C01785=1032.766,450.226,-154.652,176.488,48.489,160.264
C01786=1032.794,450.472,-154.693,176.509,48.493,160.268
C01787=1032.823,450.716,-154.734,176.528,48.497,160.272
C01788=1032.851,450.962,-154.775,176.549,48.502,160.277
C01789=1032.882,451.208,-154.815,176.569,48.506,160.281
C01790=1032.912,451.453,-154.855,176.590,48.510,160.285
C01791=1032.942,451.698,-154.894,176.611,48.514,160.290
C01792=1032.973,451.944,-154.933,176.632,48.519,160.294
C01793=1033.006,452.191,-154.972,176.652,48.523,160.299
C01794=1033.037,452.435,-155.009,176.673,48.527,160.303
C01795=1033.070,452.681,-155.047,176.695,48.530,160.307
C01796=1033.104,452.933,-155.086,176.716,48.534,160.312
C01797=1033.139,453.185,-155.123,176.737,48.538,160.316
C01798=1032.855,453.248,-155.453,176.741,48.604,160.337
C01799=1032.824,453.021,-155.419,176.721,48.600,160.333
C01800=1032.792,452.792,-155.385,176.702,48.597,160.329
C01801=1032.760,452.547,-155.347,176.680,48.593,160.325
C01802=1032.728,452.301,-155.309,176.659,48.589,160.320
C01803=1032.695,452.056,-155.271,176.639,48.585,160.316
C01804=1032.664,451.810,-155.232,176.617,48.582,160.312
C01805=1032.633,451.564,-155.193,176.596,48.578,160.307
C01806=1032.603,451.319,-155.154,176.577,48.573,160.303
C01807=1032.573,451.074,-155.114,176.556,48.569,160.299
C01808=1032.543,450.827,-155.074,176.535,48.566,160.294
C01809=1032.514,450.583,-155.033,176.515,48.561,160.290
C01810=1032.486,450.338,-154.992,176.494,48.557,160.286
C01811=1032.458,450.092,-154.950,176.474,48.552,160.281
C01812=1032.431,449.847,-154.908,176.454,48.548,160.277
C01813=1032.404,449.602,-154.865,176.434,48.543,160.273
C01814=1032.377,449.357,-154.823,176.414,48.539,160.268
C01815=1032.351,449.112,-154.779,176.394,48.534,160.264
C01816=1032.326,448.866,-154.736,176.374,48.530,160.259
C01817=1032.301,448.622,-154.691,176.355,48.524,160.255
C01818=1032.276,448.377,-154.647,176.334,48.519,160.250
C01819=1032.252,448.131,-154.602,176.316,48.515,160.246
C01820=1032.229,447.887,-154.556,176.296,48.510,160.242
C01821=1032.206,447.643,-154.511,176.276,48.504,160.237
C01822=1032.183,447.398,-154.465,176.258,48.499,160.233
C01823=1032.162,447.153,-154.418,176.238,48.494,160.228
C01824=1032.140,446.909,-154.371,176.219,48.489,160.224
C01825=1032.119,446.665,-154.324,176.200,48.483,160.220
C01826=1032.099,446.420,-154.276,176.181,48.478,160.215
C01827=1032.079,446.176,-154.227,176.162,48.472,160.211
C01828=1032.060,445.932,-154.179,176.143,48.467,160.206
C01829=1032.041,445.688,-154.130,176.124,48.461,160.201
C01830=1032.022,445.444,-154.080,176.106,48.455,160.197
C01831=1032.004,445.200,-154.030,176.088,48.449,160.193
C01832=1031.987,444.957,-153.980,176.069,48.443,160.188
C01833=1031.969,444.713,-153.928,176.050,48.437,160.183
C01834=1031.953,444.468,-153.878,176.033,48.431,160.179
C01835=1031.938,444.225,-153.826,176.014,48.425,160.174
C01836=1031.921,443.982,-153.774,175.996,48.419,160.170
C01837=1031.908,443.739,-153.721,175.977,48.412,160.165
C01838=1031.892,443.495,-153.668,175.960,48.406,160.161
C01839=1031.879,443.253,-153.615,175.942,48.399,160.156
C01840=1031.864,443.010,-153.562,175.924,48.393,160.152
C01841=1031.851,442.766,-153.509,175.906,48.386,160.147
C01842=1031.838,442.521,-153.455,175.889,48.379,160.142
C01843=1031.824,442.278,-153.402,175.870,48.374,160.138
C01844=1031.810,442.034,-153.348,175.853,48.367,160.133
C01845=1031.796,441.790,-153.296,175.836,48.361,160.129
C01846=1031.783,441.546,-153.242,175.818,48.354,160.125
C01847=1031.769,441.302,-153.190,175.801,48.347,160.120
C01848=1031.755,441.058,-153.136,175.784,48.341,160.116
C01849=1031.742,440.814,-153.084,175.766,48.335,160.111
C01850=1031.728,440.570,-153.030,175.749,48.329,160.107
C01851=1031.715,440.326,-152.977,175.732,48.322,160.103
C01852=1031.702,440.082,-152.925,175.715,48.316,160.098
C01853=1031.688,439.838,-152.871,175.698,48.310,160.094
C01854=1031.675,439.594,-152.820,175.681,48.304,160.090
C01855=1031.662,439.350,-152.766,175.664,48.297,160.085
C01856=1031.648,439.106,-152.714,175.646,48.291,160.081
C01857=1031.634,438.844,-152.657,175.629,48.284,160.076
C01858=1031.620,438.582,-152.601,175.611,48.278,160.072
C01859=1031.606,438.319,-152.544,175.593,48.271,160.067
C01860=1031.591,438.057,-152.489,175.575,48.265,160.063
C01861=1031.578,437.813,-152.436,175.559,48.258,160.059
C01862=1031.565,437.569,-152.385,175.542,48.253,160.054
C01863=1031.552,437.324,-152.332,175.526,48.246,160.050
C01864=1031.539,437.080,-152.280,175.509,48.241,160.046
C01865=1031.526,436.836,-152.228,175.494,48.234,160.042
C01866=1031.513,436.592,-152.176,175.477,48.229,160.038
C01867=1031.500,436.347,-152.124,175.461,48.222,160.034
C01868=1031.487,436.103,-152.072,175.444,48.217,160.030
C01869=1031.474,435.859,-152.021,175.429,48.211,160.026
C01870=1031.462,435.615,-151.969,175.413,48.205,160.022
C01871=1031.448,435.370,-151.917,175.396,48.199,160.018
C01872=1031.436,435.126,-151.866,175.381,48.193,160.014
C01873=1031.423,434.882,-151.814,175.365,48.187,160.010
C01874=1031.410,434.637,-151.763,175.350,48.182,160.006
C01875=1031.398,434.392,-151.711,175.334,48.176,160.002
C01876=1031.385,434.149,-151.660,175.317,48.170,159.998
C01877=1031.366,433.797,-151.586,175.296,48.162,159.992
C01878=1031.348,433.447,-151.513,175.273,48.154,159.987
C01879=1031.330,433.095,-151.440,175.251,48.145,159.981
C01880=1031.312,432.744,-151.366,175.229,48.137,159.976
C01881=1031.299,432.500,-151.315,175.214,48.132,159.972
C01882=1031.287,432.256,-151.265,175.198,48.126,159.968
C01883=1031.274,432.011,-151.214,175.183,48.121,159.965
C01884=1031.262,431.766,-151.163,175.168,48.115,159.961
C01885=1031.249,431.521,-151.112,175.153,48.110,159.957
C01886=1031.237,431.277,-151.062,175.137,48.104,159.953
C01887=1031.224,431.032,-151.011,175.123,48.098,159.950
C01888=1031.212,430.788,-150.961,175.108,48.093,159.946
C01889=1031.199,430.543,-150.910,175.093,48.087,159.942
C01890=1031.187,430.299,-150.860,175.078,48.082,159.938
C01891=1031.175,430.054,-150.809,175.064,48.077,159.935
C01892=1031.163,429.809,-150.758,175.049,48.071,159.931
C01893=1031.151,429.565,-150.709,175.033,48.066,159.928
C01894=1031.139,429.320,-150.659,175.019,48.061,159.924
C01895=1031.126,429.076,-150.608,175.004,48.055,159.920
C01896=1031.114,428.831,-150.558,174.990,48.050,159.917
C01897=1031.102,428.586,-150.507,174.976,48.045,159.913
C01898=1031.091,428.342,-150.457,174.961,48.039,159.910
C01899=1031.078,428.097,-150.407,174.946,48.034,159.906
C01900=1031.066,427.852,-150.357,174.933,48.029,159.903
C01901=1031.055,427.608,-150.308,174.919,48.023,159.899
C01902=1031.042,427.363,-150.258,174.904,48.019,159.896
C01903=1031.030,427.118,-150.208,174.890,48.013,159.892
C01904=1031.019,426.874,-150.158,174.876,48.008,159.889
C01905=1031.007,426.628,-150.108,174.861,48.003,159.885
C01906=1030.995,426.383,-150.058,174.847,47.998,159.882
C01907=1030.983,426.139,-150.009,174.834,47.993,159.878
C01908=1030.971,425.893,-149.960,174.819,47.988,159.875
C01909=1030.959,425.649,-149.911,174.805,47.983,159.872
C01910=1030.947,425.404,-149.861,174.791,47.978,159.868
C01911=1030.935,425.159,-149.812,174.778,47.972,159.865
C01912=1030.923,424.914,-149.762,174.764,47.967,159.861
C01913=1030.913,424.705,-149.720,174.752,47.963,159.859
C01914=1030.903,424.497,-149.678,174.740,47.959,159.856
C01915=1030.893,424.288,-149.636,174.729,47.955,159.853
C01916=1030.883,424.079,-149.594,174.717,47.950,159.850
C01917=1030.874,423.871,-149.553,174.706,47.947,159.847
C01918=1030.864,423.662,-149.511,174.693,47.942,159.845
C01919=1030.854,423.453,-149.469,174.682,47.938,159.842
C01920=1030.844,423.244,-149.428,174.671,47.934,159.839
C01921=1030.833,422.999,-149.379,174.657,47.929,159.836
C01922=1030.821,422.753,-149.330,174.644,47.924,159.833
C01923=1030.809,422.509,-149.280,174.630,47.920,159.829
C01924=1030.797,422.264,-149.233,174.617,47.914,159.826
C01925=1030.786,422.019,-149.184,174.604,47.910,159.823
C01926=1030.775,421.773,-149.135,174.591,47.905,159.820
C01927=1030.763,421.529,-149.087,174.578,47.900,159.817
C01928=1030.751,421.283,-149.038,174.564,47.896,159.813
C01929=1030.740,421.038,-148.989,174.551,47.891,159.810
C01930=1030.729,420.793,-148.941,174.539,47.886,159.807
C01931=1030.717,420.548,-148.893,174.525,47.882,159.804
C01932=1030.705,420.303,-148.844,174.512,47.877,159.801
C01933=1030.695,420.058,-148.796,174.499,47.872,159.798
C01934=1030.683,419.813,-148.749,174.486,47.867,159.795
C01935=1030.672,419.568,-148.700,174.473,47.863,159.792
C01936=1030.661,419.323,-148.652,174.461,47.858,159.789
C01937=1030.649,419.078,-148.604,174.447,47.854,159.786
C01938=1030.638,418.832,-148.556,174.434,47.850,159.783
C01939=1030.627,418.587,-148.508,174.422,47.845,159.779
C01940=1030.616,418.342,-148.461,174.409,47.841,159.777
C01941=1030.604,418.097,-148.412,174.397,47.836,159.773
C01942=1030.593,417.852,-148.364,174.384,47.831,159.771
C01943=1030.582,417.607,-148.317,174.372,47.827,159.768
C01944=1030.571,417.361,-148.269,174.359,47.822,159.765
C01945=1030.560,417.116,-148.221,174.346,47.818,159.762
C01946=1030.549,416.872,-148.173,174.334,47.814,159.759
C01947=1030.538,416.626,-148.126,174.322,47.809,159.756
C01948=1030.527,416.380,-148.077,174.310,47.805,159.753
C01949=1030.516,416.135,-148.031,174.298,47.801,159.750
C01950=1030.505,415.890,-147.983,174.285,47.796,159.747
C01951=1030.494,415.645,-147.936,174.273,47.792,159.744
C01952=1030.483,415.399,-147.889,174.261,47.788,159.741
C01953=1030.472,415.154,-147.842,174.248,47.783,159.739
C01954=1030.461,414.909,-147.794,174.236,47.780,159.736
C01955=1030.450,414.664,-147.747,174.224,47.775,159.733
C01956=1030.439,414.418,-147.700,174.212,47.771,159.730
C01957=1030.428,414.173,-147.653,174.199,47.767,159.727
C01958=1030.418,413.928,-147.606,174.187,47.763,159.725
C01959=1030.406,413.682,-147.559,174.175,47.758,159.722
C01960=1030.396,413.437,-147.512,174.164,47.754,159.719
C01961=1030.385,413.192,-147.465,174.152,47.750,159.716
C01962=1030.374,412.947,-147.419,174.140,47.746,159.713
C01963=1030.363,412.701,-147.371,174.128,47.742,159.711
C01964=1030.352,412.456,-147.324,174.116,47.737,159.708
C01965=1030.343,412.210,-147.278,174.105,47.733,159.705
C01966=1030.332,411.965,-147.231,174.093,47.730,159.703
C01967=1030.321,411.720,-147.185,174.082,47.726,159.700
C01968=1030.310,411.473,-147.138,174.070,47.722,159.697
C01969=1030.299,411.229,-147.091,174.058,47.717,159.694
C01970=1030.289,410.983,-147.044,174.046,47.713,159.692
C01971=1030.278,410.738,-146.998,174.035,47.709,159.689
C01972=1030.268,410.492,-146.951,174.023,47.705,159.686
C01973=1030.258,410.247,-146.905,174.012,47.702,159.684
C01974=1030.247,410.001,-146.859,174.000,47.698,159.681
C01975=1030.236,409.756,-146.813,173.989,47.694,159.679
C01976=1030.226,409.510,-146.767,173.977,47.690,159.676
C01977=1030.215,409.241,-146.716,173.965,47.686,159.673
C01978=1030.203,408.972,-146.666,173.952,47.682,159.670
C01979=1030.191,408.703,-146.615,173.940,47.677,159.668
C01980=1030.180,408.433,-146.565,173.928,47.674,159.665
C01981=1030.169,408.188,-146.519,173.916,47.670,159.662
C01982=1030.158,407.942,-146.473,173.906,47.666,159.660
C01983=1030.148,407.696,-146.428,173.894,47.662,159.657
C01984=1030.137,407.451,-146.382,173.883,47.659,159.655
C01985=1030.127,407.205,-146.336,173.871,47.655,159.652
C01986=1030.117,406.960,-146.290,173.861,47.651,159.650
C01987=1030.106,406.715,-146.244,173.850,47.648,159.647
C01988=1030.096,406.468,-146.198,173.838,47.644,159.645
C01989=1030.086,406.223,-146.153,173.828,47.640,159.642
C01990=1030.076,405.978,-146.107,173.817,47.637,159.640
C01991=1030.065,405.732,-146.062,173.806,47.633,159.637
C01992=1030.055,405.487,-146.016,173.795,47.629,159.635
C01993=1030.045,405.240,-145.971,173.784,47.626,159.633
C01994=1030.035,404.996,-145.926,173.773,47.622,159.630
C01995=1030.025,404.749,-145.880,173.762,47.619,159.628
C01996=1030.015,404.504,-145.835,173.752,47.615,159.625
C01997=1030.004,404.258,-145.790,173.741,47.612,159.623
C01998=1029.994,404.013,-145.744,173.730,47.608,159.620
C01999=1029.984,403.767,-145.699,173.719,47.605,159.618
C02000=1029.974,403.522,-145.654,173.709,47.601,159.616
C02001=1029.964,403.276,-145.608,173.699,47.598,159.613
C02002=1029.954,403.031,-145.563,173.688,47.594,159.611
C02003=1029.944,402.785,-145.519,173.677,47.590,159.609
C02004=1029.934,402.539,-145.473,173.666,47.588,159.606
C02005=1029.924,402.293,-145.429,173.656,47.584,159.604
C02006=1029.915,402.048,-145.384,173.646,47.581,159.602
C02007=1029.904,401.802,-145.339,173.635,47.577,159.599
C02008=1029.894,401.556,-145.294,173.625,47.574,159.597
C02009=1029.885,401.311,-145.249,173.615,47.570,159.595
C02010=1029.874,401.064,-145.204,173.604,47.567,159.593
C02011=1029.865,400.819,-145.159,173.594,47.564,159.590
C02012=1029.855,400.573,-145.114,173.583,47.560,159.588
C02013=1029.846,400.327,-145.070,173.573,47.557,159.586
C02014=1029.835,400.082,-145.026,173.563,47.554,159.584
C02015=1029.825,399.836,-144.981,173.552,47.550,159.581
C02016=1029.815,399.590,-144.936,173.542,47.547,159.579
C02017=1029.806,399.344,-144.892,173.531,47.544,159.577
C02018=1029.795,399.099,-144.847,173.521,47.541,159.575
C02019=1029.786,398.853,-144.803,173.512,47.538,159.572
C02020=1029.776,398.607,-144.758,173.502,47.535,159.570
C02021=1029.767,398.361,-144.714,173.492,47.532,159.568
C02022=1029.757,398.115,-144.671,173.482,47.528,159.566
C02023=1029.747,397.870,-144.626,173.471,47.525,159.564
C02024=1029.737,397.624,-144.582,173.461,47.523,159.562
C02025=1029.727,397.378,-144.538,173.451,47.520,159.560
C02026=1029.718,397.132,-144.494,173.441,47.516,159.557
C02027=1029.707,396.886,-144.450,173.431,47.513,159.555
C02028=1029.698,396.640,-144.406,173.422,47.510,159.553
C02029=1029.689,396.394,-144.362,173.412,47.507,159.551
C02030=1029.678,396.148,-144.318,173.402,47.504,159.549
C02031=1029.670,395.903,-144.275,173.392,47.501,159.547
C02032=1029.660,395.657,-144.230,173.382,47.498,159.545
C02033=1029.650,395.411,-144.187,173.373,47.495,159.543
C02034=1029.641,395.165,-144.143,173.363,47.492,159.541
C02035=1029.631,394.919,-144.099,173.353,47.490,159.539
C02036=1029.622,394.674,-144.056,173.343,47.486,159.536
C02037=1029.611,394.425,-144.011,173.334,47.484,159.534
C02038=1029.602,394.178,-143.967,173.324,47.480,159.532
C02039=1029.593,393.930,-143.923,173.314,47.478,159.530
C02040=1029.583,393.683,-143.880,173.304,47.475,159.528
C02041=1029.574,393.436,-143.836,173.295,47.472,159.526
C02042=1029.564,393.190,-143.793,173.285,47.469,159.524
C02043=1029.555,392.944,-143.750,173.276,47.467,159.522
C02044=1029.545,392.698,-143.706,173.266,47.464,159.520
C02045=1029.535,392.452,-143.663,173.256,47.461,159.518
C02046=1029.527,392.206,-143.620,173.247,47.459,159.516
C02047=1029.517,391.960,-143.577,173.238,47.455,159.514
C02048=1029.508,391.714,-143.533,173.228,47.452,159.512
C02049=1029.498,391.468,-143.490,173.219,47.450,159.510
C02050=1029.489,391.223,-143.446,173.209,47.447,159.508
C02051=1029.479,390.976,-143.404,173.200,47.445,159.506
C02052=1029.470,390.730,-143.361,173.191,47.442,159.505
C02053=1029.461,390.484,-143.317,173.182,47.439,159.503
C02054=1029.452,390.239,-143.275,173.172,47.436,159.501
C02055=1029.442,389.992,-143.231,173.162,47.434,159.499
C02056=1029.433,389.746,-143.189,173.154,47.431,159.497
C02057=1029.423,389.500,-143.146,173.145,47.429,159.495
C02058=1029.415,389.254,-143.103,173.135,47.426,159.493
C02059=1029.405,389.007,-143.060,173.126,47.423,159.491
C02060=1029.396,388.761,-143.018,173.117,47.421,159.489
C02061=1029.387,388.516,-142.975,173.108,47.418,159.487
C02062=1029.377,388.269,-142.932,173.098,47.416,159.486
C02063=1029.368,388.023,-142.890,173.090,47.413,159.484
C02064=1029.359,387.777,-142.847,173.080,47.411,159.482
C02065=1029.350,387.531,-142.804,173.072,47.408,159.480
C02066=1029.341,387.285,-142.761,173.063,47.406,159.478
C02067=1029.332,387.038,-142.720,173.053,47.403,159.476
C02068=1029.322,386.793,-142.677,173.045,47.401,159.475
C02069=1029.313,386.546,-142.634,173.036,47.399,159.473
C02070=1029.304,386.300,-142.592,173.027,47.396,159.471
C02071=1029.295,386.054,-142.550,173.018,47.393,159.469
C02072=1029.286,385.807,-142.508,173.008,47.391,159.467
C02073=1029.276,385.561,-142.465,173.000,47.389,159.466
C02074=1029.267,385.315,-142.423,172.991,47.387,159.464
C02075=1029.258,385.069,-142.381,172.983,47.384,159.462
C02076=1029.249,384.823,-142.339,172.973,47.382,159.460
C02077=1029.240,384.576,-142.298,172.965,47.380,159.459
C02078=1029.231,384.330,-142.255,172.956,47.377,159.457
C02079=1029.222,384.084,-142.213,172.948,47.375,159.455
C02080=1029.213,383.838,-142.172,172.938,47.373,159.453
C02081=1029.203,383.591,-142.129,172.930,47.371,159.452
C02082=1029.194,383.345,-142.087,172.921,47.368,159.450
C02083=1029.186,383.099,-142.045,172.913,47.366,159.448
C02084=1029.177,382.852,-142.004,172.903,47.364,159.446
C02085=1029.168,382.606,-141.962,172.895,47.361,159.445
C02086=1029.159,382.359,-141.920,172.887,47.359,159.443
C02087=1029.150,382.113,-141.879,172.878,47.357,159.442
C02088=1029.141,381.867,-141.837,172.870,47.355,159.440
C02089=1029.133,381.621,-141.795,172.860,47.353,159.438
C02090=1029.124,381.375,-141.754,172.852,47.350,159.436
C02091=1029.115,381.128,-141.712,172.844,47.348,159.435
C02092=1029.106,380.882,-141.670,172.835,47.346,159.433
C02093=1029.097,380.653,-141.631,172.827,47.344,159.432
C02094=1029.089,380.424,-141.593,172.819,47.343,159.430
C02095=1029.081,380.196,-141.554,172.812,47.340,159.429
C02096=1029.072,379.967,-141.516,172.804,47.339,159.427
C02097=1029.065,379.737,-141.478,172.796,47.337,159.426
C02098=1029.056,379.509,-141.439,172.788,47.335,159.424
C02099=1029.048,379.279,-141.401,172.780,47.332,159.422
C02100=1029.040,379.050,-141.362,172.772,47.331,159.421
C02101=1029.031,378.804,-141.321,172.764,47.329,159.419
C02102=1029.022,378.557,-141.279,172.756,47.327,159.418
C02103=1029.014,378.311,-141.238,172.748,47.324,159.416
C02104=1029.005,378.065,-141.197,172.739,47.323,159.415
C02105=1028.996,377.818,-141.155,172.731,47.321,159.413
C02106=1028.988,377.572,-141.114,172.723,47.318,159.411
C02107=1028.979,377.326,-141.073,172.715,47.317,159.410
C02108=1028.971,377.079,-141.032,172.707,47.315,159.408
C02109=1028.962,376.832,-140.991,172.698,47.313,159.407
C02110=1028.953,376.586,-140.950,172.690,47.311,159.405
C02111=1028.944,376.339,-140.909,172.682,47.309,159.404
C02112=1028.936,376.094,-140.869,172.674,47.307,159.402
C02113=1028.927,375.847,-140.828,172.666,47.306,159.401
C02114=1028.918,375.600,-140.787,172.658,47.304,159.399
C02115=1028.909,375.354,-140.746,172.650,47.302,159.398
C02116=1028.901,375.107,-140.705,172.642,47.300,159.396
C02117=1028.893,374.861,-140.664,172.634,47.298,159.395
C02118=1028.883,374.614,-140.624,172.626,47.296,159.393
C02119=1028.875,374.368,-140.583,172.618,47.294,159.392
C02120=1028.867,374.121,-140.542,172.610,47.293,159.390
C02121=1028.858,373.875,-140.502,172.602,47.291,159.389
C02122=1028.849,373.628,-140.461,172.594,47.289,159.387
C02123=1028.840,373.382,-140.421,172.586,47.288,159.386
C02124=1028.832,373.135,-140.380,172.578,47.286,159.384
C02125=1028.824,372.889,-140.340,172.570,47.284,159.383
C02126=1028.815,372.641,-140.300,172.562,47.282,159.381
C02127=1028.807,372.395,-140.259,172.554,47.281,159.380
C02128=1028.799,372.149,-140.219,172.546,47.279,159.378
C02129=1028.789,371.902,-140.178,172.538,47.277,159.377
C02130=1028.781,371.656,-140.138,172.531,47.276,159.376
C02131=1028.774,371.409,-140.098,172.523,47.274,159.374
C02132=1028.764,371.162,-140.057,172.515,47.273,159.373
C02133=1028.756,370.916,-140.017,172.507,47.271,159.371
C02134=1028.748,370.669,-139.977,172.500,47.269,159.370
C02135=1028.740,370.423,-139.937,172.492,47.267,159.368
C02136=1028.731,370.176,-139.896,172.484,47.266,159.367
C02137=1028.723,369.930,-139.856,172.476,47.264,159.366
C02138=1028.715,369.683,-139.816,172.469,47.263,159.364
C02139=1028.706,369.437,-139.776,172.462,47.261,159.363
C02140=1028.698,369.190,-139.736,172.454,47.259,159.361
C02141=1028.690,368.943,-139.696,172.447,47.258,159.360
C02142=1028.681,368.696,-139.656,172.439,47.256,159.359
C02143=1028.673,368.450,-139.616,172.431,47.255,159.357
C02144=1028.665,368.203,-139.576,172.423,47.253,159.356
C02145=1028.656,367.956,-139.537,172.416,47.252,159.355
C02146=1028.647,367.709,-139.497,172.408,47.251,159.353
C02147=1028.639,367.463,-139.458,172.400,47.249,159.352
C02148=1028.631,367.217,-139.417,172.393,47.248,159.351
C02149=1028.622,366.970,-139.378,172.385,47.246,159.349
C02150=1028.614,366.723,-139.339,172.378,47.245,159.348
C02151=1028.606,366.477,-139.299,172.371,47.243,159.347
C02152=1028.598,366.230,-139.259,172.363,47.242,159.345
C02153=1028.590,366.011,-139.225,172.357,47.241,159.344
C02154=1028.583,365.792,-139.189,172.350,47.239,159.343
C02155=1028.575,365.574,-139.155,172.343,47.239,159.342
C02156=1028.568,365.356,-139.120,172.337,47.238,159.341
C02157=1028.561,365.137,-139.084,172.330,47.236,159.340
C02158=1028.553,364.919,-139.049,172.324,47.235,159.339
C02159=1028.546,364.701,-139.015,172.317,47.233,159.337
C02160=1028.539,364.482,-138.980,172.311,47.232,159.336
C02161=1028.531,364.235,-138.940,172.303,47.231,159.335
C02162=1028.522,363.988,-138.901,172.296,47.230,159.334
C02163=1028.515,363.742,-138.861,172.289,47.229,159.333
C02164=1028.506,363.494,-138.823,172.282,47.227,159.331
C02165=1028.498,363.248,-138.783,172.274,47.226,159.330
C02166=1028.490,363.002,-138.744,172.267,47.225,159.329
C02167=1028.483,362.754,-138.705,172.260,47.224,159.328
C02168=1028.474,362.508,-138.666,172.253,47.222,159.326
C02169=1028.466,362.261,-138.627,172.245,47.221,159.325
C02170=1028.458,362.014,-138.587,172.238,47.220,159.324
C02171=1028.450,361.767,-138.548,172.231,47.219,159.323
C02172=1028.442,361.521,-138.509,172.224,47.217,159.321
C02173=1028.434,361.274,-138.470,172.217,47.217,159.320
C02174=1028.426,361.027,-138.430,172.210,47.215,159.319
C02175=1028.418,360.780,-138.392,172.203,47.214,159.318
C02176=1028.410,360.533,-138.353,172.195,47.213,159.316
C02177=1028.402,360.287,-138.314,172.189,47.212,159.315
C02178=1028.394,360.039,-138.276,172.181,47.211,159.314
C02179=1028.385,359.793,-138.236,172.174,47.210,159.313
C02180=1028.377,359.546,-138.198,172.167,47.208,159.312
C02181=1028.370,359.299,-138.160,172.160,47.207,159.311
C02182=1028.362,359.052,-138.121,172.153,47.207,159.309
C02183=1028.353,358.805,-138.082,172.146,47.205,159.308
C02184=1028.346,358.559,-138.043,172.139,47.204,159.307
C02185=1028.337,358.312,-138.005,172.132,47.204,159.306
C02186=1028.329,358.064,-137.966,172.125,47.202,159.305
C02187=1028.322,357.818,-137.928,172.118,47.201,159.304
C02188=1028.314,357.571,-137.889,172.111,47.200,159.303
C02189=1028.305,357.323,-137.851,172.104,47.199,159.301
C02190=1028.298,357.077,-137.812,172.097,47.199,159.300
C02191=1028.290,356.830,-137.774,172.091,47.198,159.299
C02192=1028.282,356.583,-137.736,172.083,47.196,159.298
C02193=1028.273,356.336,-137.698,172.077,47.195,159.297
C02194=1028.265,356.089,-137.659,172.069,47.195,159.296
C02195=1028.258,355.843,-137.621,172.063,47.193,159.295
C02196=1028.249,355.595,-137.582,172.056,47.193,159.294
C02197=1028.242,355.349,-137.544,172.050,47.192,159.293
C02198=1028.234,355.102,-137.505,172.042,47.191,159.291
C02199=1028.226,354.854,-137.468,172.036,47.190,159.290
C02200=1028.218,354.607,-137.429,172.029,47.189,159.289
C02201=1028.210,354.361,-137.391,172.021,47.188,159.288
C02202=1028.202,354.114,-137.353,172.015,47.187,159.287
C02203=1028.195,353.867,-137.315,172.008,47.187,159.286
C02204=1028.186,353.619,-137.277,172.002,47.186,159.285
C02205=1028.178,353.373,-137.240,171.995,47.185,159.284
C02206=1028.171,353.126,-137.202,171.988,47.184,159.283
C02207=1028.163,352.879,-137.163,171.981,47.184,159.282
C02208=1028.156,352.632,-137.125,171.975,47.183,159.281
C02209=1028.147,352.385,-137.087,171.968,47.182,159.280
C02210=1028.139,352.138,-137.050,171.962,47.181,159.279
C02211=1028.132,351.891,-137.012,171.955,47.180,159.278
C02212=1028.124,351.643,-136.974,171.948,47.180,159.277
C02213=1028.117,351.429,-136.941,171.942,47.179,159.276
C02214=1028.111,351.213,-136.908,171.937,47.178,159.275
C02215=1028.103,350.998,-136.875,171.931,47.178,159.274
C02216=1028.097,350.782,-136.842,171.925,47.178,159.273
C02217=1028.090,350.568,-136.810,171.919,47.177,159.272
C02218=1028.083,350.352,-136.777,171.914,47.176,159.271
C02219=1028.076,350.137,-136.744,171.908,47.175,159.270
C02220=1028.070,349.922,-136.711,171.902,47.175,159.269
C02221=1028.063,349.675,-136.673,171.896,47.174,159.269
C02222=1028.054,349.428,-136.636,171.890,47.173,159.268
C02223=1028.047,349.180,-136.598,171.882,47.173,159.266
C02224=1028.040,348.933,-136.561,171.877,47.172,159.266
C02225=1028.032,348.686,-136.524,171.870,47.172,159.265
C02226=1028.024,348.440,-136.485,171.863,47.171,159.264
C02227=1028.015,348.192,-136.448,171.857,47.171,159.263
C02228=1028.008,347.945,-136.411,171.850,47.170,159.262
C02229=1028.000,347.698,-136.374,171.844,47.169,159.261
C02230=1027.993,347.451,-136.336,171.838,47.169,159.260
C02231=1027.985,347.204,-136.299,171.831,47.168,159.259
C02232=1027.977,346.957,-136.261,171.825,47.168,159.258
C02233=1027.969,346.710,-136.224,171.819,47.167,159.257
C02234=1027.962,346.463,-136.187,171.812,47.166,159.256
C02235=1027.954,346.215,-136.151,171.806,47.166,159.255
C02236=1027.947,345.968,-136.113,171.800,47.166,159.254
C02237=1027.939,345.721,-136.076,171.793,47.165,159.253
C02238=1027.932,345.474,-136.039,171.787,47.165,159.252
C02239=1027.924,345.227,-136.002,171.780,47.164,159.251
C02240=1027.917,344.980,-135.964,171.774,47.164,159.250
C02241=1027.909,344.733,-135.928,171.768,47.163,159.249
C02242=1027.901,344.486,-135.891,171.762,47.163,159.249
C02243=1027.894,344.239,-135.854,171.755,47.163,159.248
C02244=1027.886,343.991,-135.817,171.749,47.162,159.247
C02245=1027.879,343.744,-135.780,171.743,47.162,159.246
C02246=1027.871,343.497,-135.743,171.737,47.161,159.245
C02247=1027.864,343.250,-135.706,171.730,47.161,159.244
C02248=1027.856,343.003,-135.669,171.724,47.161,159.243
C02249=1027.848,342.755,-135.633,171.718,47.160,159.242
C02250=1027.841,342.508,-135.595,171.712,47.160,159.241
C02251=1027.833,342.261,-135.558,171.705,47.160,159.241
C02252=1027.825,342.014,-135.522,171.699,47.159,159.240
C02253=1027.818,341.766,-135.485,171.693,47.159,159.239
C02254=1027.810,341.519,-135.448,171.687,47.158,159.238
C02255=1027.803,341.272,-135.412,171.681,47.158,159.237
C02256=1027.795,341.025,-135.375,171.674,47.158,159.236
C02257=1027.788,340.777,-135.339,171.668,47.157,159.235
C02258=1027.780,340.531,-135.302,171.662,47.157,159.234
C02259=1027.773,340.283,-135.265,171.656,47.157,159.234
C02260=1027.766,340.036,-135.229,171.651,47.156,159.233
C02261=1027.758,339.789,-135.193,171.644,47.156,159.232
C02262=1027.750,339.542,-135.156,171.638,47.156,159.231
C02263=1027.742,339.294,-135.120,171.632,47.156,159.230
C02264=1027.735,339.048,-135.084,171.626,47.155,159.229
C02265=1027.728,338.800,-135.047,171.620,47.155,159.229
C02266=1027.721,338.552,-135.011,171.613,47.155,159.228
C02267=1027.713,338.305,-134.974,171.607,47.155,159.227
C02268=1027.705,338.057,-134.938,171.602,47.155,159.226
C02269=1027.698,337.811,-134.902,171.596,47.155,159.225
C02270=1027.690,337.564,-134.865,171.590,47.154,159.225
C02271=1027.683,337.316,-134.829,171.584,47.154,159.224
C02272=1027.675,337.069,-134.793,171.577,47.154,159.223
C02273=1027.669,336.852,-134.762,171.573,47.154,159.222
C02274=1027.662,336.636,-134.730,171.567,47.154,159.222
C02275=1027.656,336.418,-134.698,171.562,47.154,159.221
C02276=1027.649,336.202,-134.667,171.556,47.154,159.220
C02277=1027.643,335.985,-134.634,171.552,47.153,159.219
C02278=1027.637,335.768,-134.604,171.546,47.154,159.219
C02279=1027.630,335.552,-134.571,171.541,47.154,159.218
C02280=1027.624,335.334,-134.540,171.536,47.154,159.217
C02281=1027.616,335.087,-134.504,171.530,47.153,159.217
C02282=1027.610,334.840,-134.468,171.524,47.153,159.216
C02283=1027.602,334.592,-134.432,171.518,47.154,159.215
C02284=1027.595,334.346,-134.396,171.512,47.153,159.214
C02285=1027.587,334.098,-134.360,171.507,47.153,159.214
C02286=1027.580,333.850,-134.324,171.501,47.153,159.213
C02287=1027.573,333.603,-134.288,171.495,47.153,159.212
C02288=1027.565,333.355,-134.253,171.490,47.153,159.211
C02289=1027.558,333.109,-134.217,171.484,47.153,159.211
C02290=1027.550,332.861,-134.181,171.478,47.153,159.210
C02291=1027.543,332.614,-134.146,171.472,47.153,159.209
C02292=1027.535,332.367,-134.110,171.466,47.153,159.208
C02293=1027.529,332.119,-134.075,171.460,47.153,159.208
C02294=1027.521,331.872,-134.038,171.454,47.154,159.207
C02295=1027.514,331.624,-134.003,171.449,47.154,159.206
C02296=1027.506,331.377,-133.968,171.443,47.153,159.205
C02297=1027.499,331.130,-133.933,171.437,47.153,159.205
C02298=1027.491,330.883,-133.896,171.431,47.154,159.204
C02299=1027.485,330.635,-133.861,171.426,47.154,159.203
C02300=1027.477,330.388,-133.825,171.420,47.154,159.203
C02301=1027.470,330.140,-133.790,171.414,47.154,159.202
C02302=1027.462,329.893,-133.755,171.409,47.154,159.201
C02303=1027.455,329.646,-133.719,171.403,47.154,159.201
C02304=1027.448,329.398,-133.684,171.397,47.154,159.200
C02305=1027.441,329.150,-133.648,171.392,47.155,159.199
C02306=1027.434,328.904,-133.613,171.386,47.155,159.199
C02307=1027.426,328.656,-133.578,171.380,47.155,159.198
C02308=1027.419,328.409,-133.543,171.375,47.155,159.197
C02309=1027.412,328.161,-133.507,171.369,47.155,159.197
C02310=1027.404,327.914,-133.471,171.363,47.155,159.196
C02311=1027.398,327.666,-133.436,171.358,47.155,159.195
C02312=1027.390,327.419,-133.402,171.352,47.156,159.194
C02313=1027.383,327.171,-133.366,171.347,47.156,159.194
C02314=1027.375,326.924,-133.332,171.341,47.157,159.193
C02315=1027.368,326.677,-133.296,171.336,47.157,159.193
C02316=1027.360,326.429,-133.261,171.330,47.157,159.192
C02317=1027.353,326.182,-133.227,171.325,47.158,159.191
C02318=1027.346,325.935,-133.192,171.319,47.158,159.191
C02319=1027.338,325.687,-133.157,171.313,47.158,159.190
C02320=1027.331,325.440,-133.122,171.308,47.159,159.190
C02321=1027.324,325.192,-133.088,171.302,47.159,159.189
C02322=1027.316,324.944,-133.053,171.297,47.159,159.188
C02323=1027.309,324.697,-133.018,171.291,47.160,159.188
C02324=1027.302,324.450,-132.983,171.286,47.160,159.187
C02325=1027.295,324.202,-132.948,171.280,47.161,159.186
C02326=1027.287,323.954,-132.914,171.275,47.161,159.186
C02327=1027.280,323.707,-132.880,171.269,47.161,159.185
C02328=1027.273,323.460,-132.844,171.264,47.162,159.185
C02329=1027.265,323.213,-132.810,171.258,47.162,159.184
C02330=1027.259,322.965,-132.775,171.253,47.163,159.183
C02331=1027.251,322.717,-132.741,171.247,47.163,159.183
C02332=1027.243,322.470,-132.706,171.243,47.163,159.182
C02333=1027.237,322.250,-132.675,171.237,47.163,159.182
C02334=1027.231,322.031,-132.644,171.233,47.164,159.181
C02335=1027.224,321.812,-132.614,171.227,47.165,159.181
C02336=1027.218,321.593,-132.584,171.223,47.165,159.180
C02337=1027.211,321.374,-132.553,171.218,47.165,159.180
C02338=1027.205,321.155,-132.522,171.213,47.166,159.179
C02339=1027.200,320.936,-132.492,171.209,47.166,159.179
C02340=1027.192,320.718,-132.462,171.204,47.167,159.178
C02341=1027.186,320.470,-132.427,171.199,47.167,159.177
C02342=1027.179,320.223,-132.393,171.193,47.168,159.177
C02343=1027.171,319.975,-132.359,171.188,47.168,159.176
C02344=1027.164,319.727,-132.323,171.182,47.168,159.176
C02345=1027.157,319.479,-132.290,171.177,47.169,159.175
C02346=1027.150,319.232,-132.254,171.171,47.169,159.175
C02347=1027.143,318.984,-132.221,171.167,47.170,159.174
C02348=1027.136,318.736,-132.187,171.162,47.171,159.174
C02349=1027.129,318.489,-132.152,171.156,47.171,159.173
C02350=1027.122,318.241,-132.118,171.150,47.171,159.172
C02351=1027.114,317.994,-132.083,171.145,47.172,159.172
C02352=1027.108,317.747,-132.049,171.140,47.173,159.171
C02353=1027.101,317.499,-132.015,171.135,47.173,159.171
C02354=1027.094,317.252,-131.981,171.130,47.174,159.170
C02355=1027.087,317.004,-131.946,171.124,47.174,159.170
C02356=1027.080,316.757,-131.913,171.119,47.175,159.169
C02357=1027.073,316.509,-131.879,171.113,47.175,159.169
C02358=1027.066,316.262,-131.844,171.108,47.176,159.168
C02359=1027.059,316.014,-131.810,171.104,47.176,159.168
C02360=1027.052,315.766,-131.776,171.098,47.177,159.167
C02361=1027.046,315.519,-131.742,171.093,47.178,159.167
C02362=1027.038,315.272,-131.707,171.088,47.179,159.166
C02363=1027.031,315.024,-131.674,171.082,47.180,159.166
C02364=1027.024,314.776,-131.639,171.078,47.179,159.165
C02365=1027.017,314.529,-131.605,171.072,47.180,159.164
C02366=1027.010,314.281,-131.572,171.067,47.181,159.164
C02367=1027.004,314.034,-131.537,171.062,47.182,159.163
C02368=1026.997,313.786,-131.504,171.057,47.182,159.163
C02369=1026.990,313.538,-131.470,171.052,47.183,159.162
C02370=1026.983,313.291,-131.435,171.047,47.184,159.162
C02371=1026.976,313.044,-131.401,171.041,47.184,159.161
C02372=1026.969,312.796,-131.367,171.037,47.185,159.161
C02373=1026.963,312.548,-131.333,171.032,47.186,159.160
C02374=1026.956,312.301,-131.299,171.026,47.186,159.160
C02375=1026.949,312.054,-131.266,171.021,47.187,159.159
C02376=1026.943,311.806,-131.231,171.017,47.188,159.159
C02377=1026.935,311.558,-131.197,171.011,47.188,159.158
C02378=1026.929,311.311,-131.164,171.006,47.189,159.158
C02379=1026.922,311.063,-131.131,171.000,47.190,159.157
C02380=1026.916,310.816,-131.097,170.996,47.190,159.157
C02381=1026.909,310.568,-131.063,170.991,47.191,159.157
C02382=1026.901,310.321,-131.030,170.986,47.193,159.156
C02383=1026.894,310.072,-130.997,170.980,47.193,159.156
C02384=1026.887,309.825,-130.963,170.976,47.194,159.155
C02385=1026.879,309.578,-130.930,170.971,47.195,159.155
C02386=1026.873,309.330,-130.897,170.966,47.196,159.154
C02387=1026.866,309.083,-130.863,170.960,47.197,159.154
C02388=1026.858,308.835,-130.831,170.955,47.198,159.154
C02389=1026.851,308.587,-130.797,170.951,47.199,159.153
C02390=1026.845,308.339,-130.764,170.946,47.200,159.153
C02391=1026.837,308.092,-130.731,170.941,47.201,159.152
C02392=1026.830,307.844,-130.698,170.935,47.201,159.152
C02393=1026.824,307.628,-130.669,170.931,47.203,159.152
C02394=1026.817,307.411,-130.640,170.927,47.203,159.151
C02395=1026.812,307.194,-130.611,170.923,47.204,159.151
C02396=1026.805,306.977,-130.582,170.918,47.205,159.150
C02397=1026.799,306.761,-130.553,170.914,47.206,159.150
C02398=1026.794,306.545,-130.524,170.909,47.207,159.150
C02399=1026.787,306.328,-130.495,170.905,47.208,159.149
C02400=1026.781,306.112,-130.466,170.901,47.209,159.149
C02401=1026.774,305.864,-130.434,170.896,47.209,159.149
C02402=1026.767,305.617,-130.400,170.892,47.211,159.148
C02403=1026.760,305.368,-130.367,170.886,47.211,159.148
C02404=1026.753,305.121,-130.335,170.881,47.213,159.147
C02405=1026.746,304.873,-130.301,170.877,47.213,159.147
C02406=1026.740,304.626,-130.268,170.872,47.215,159.147
C02407=1026.732,304.378,-130.236,170.867,47.215,159.146
C02408=1026.726,304.130,-130.203,170.861,47.217,159.146
C02409=1026.719,303.883,-130.169,170.857,47.218,159.146
C02410=1026.712,303.635,-130.137,170.852,47.219,159.145
C02411=1026.705,303.387,-130.104,170.847,47.220,159.145
C02412=1026.698,303.139,-130.071,170.843,47.220,159.144
C02413=1026.691,302.891,-130.039,170.838,47.222,159.144
C02414=1026.684,302.644,-130.005,170.833,47.223,159.144
C02415=1026.677,302.396,-129.972,170.828,47.224,159.143
C02416=1026.670,302.149,-129.940,170.823,47.225,159.143
C02417=1026.664,301.901,-129.907,170.818,47.226,159.142
C02418=1026.657,301.653,-129.874,170.814,47.227,159.142
C02419=1026.650,301.406,-129.842,170.809,47.228,159.142
C02420=1026.643,301.157,-129.809,170.804,47.230,159.141
C02421=1026.637,300.910,-129.776,170.800,47.231,159.141
C02422=1026.630,300.662,-129.744,170.794,47.232,159.141
C02423=1026.623,300.414,-129.711,170.789,47.233,159.140
C02424=1026.617,300.167,-129.678,170.785,47.234,159.140
C02425=1026.610,299.919,-129.646,170.780,47.235,159.140
C02426=1026.603,299.671,-129.613,170.776,47.236,159.139
C02427=1026.596,299.423,-129.580,170.771,47.237,159.139
C02428=1026.589,299.176,-129.548,170.766,47.239,159.139
C02429=1026.582,298.928,-129.515,170.762,47.240,159.138
C02430=1026.576,298.680,-129.482,170.757,47.241,159.138
C02431=1026.569,298.433,-129.450,170.751,47.242,159.137
C02432=1026.562,298.185,-129.417,170.747,47.243,159.137
C02433=1026.556,297.937,-129.384,170.742,47.244,159.137
C02434=1026.549,297.690,-129.352,170.738,47.246,159.137
C02435=1026.543,297.442,-129.320,170.733,47.247,159.136
C02436=1026.536,297.193,-129.287,170.728,47.248,159.136
C02437=1026.529,296.946,-129.255,170.724,47.249,159.136
C02438=1026.523,296.698,-129.222,170.719,47.250,159.135
C02439=1026.516,296.451,-129.190,170.715,47.251,159.135
C02440=1026.510,296.203,-129.158,170.710,47.253,159.135
C02441=1026.503,295.955,-129.125,170.706,47.254,159.134
C02442=1026.496,295.707,-129.092,170.701,47.255,159.134
C02443=1026.489,295.460,-129.060,170.696,47.257,159.134
C02444=1026.483,295.212,-129.028,170.692,47.258,159.133
C02445=1026.476,294.964,-128.996,170.687,47.259,159.133
C02446=1026.470,294.717,-128.963,170.682,47.260,159.133
C02447=1026.464,294.468,-128.930,170.677,47.262,159.132
C02448=1026.457,294.220,-128.898,170.673,47.263,159.132
C02449=1026.450,293.973,-128.866,170.668,47.264,159.132
C02450=1026.444,293.725,-128.834,170.664,47.265,159.131
C02451=1026.437,293.478,-128.802,170.659,47.267,159.131
C02452=1026.431,293.229,-128.770,170.654,47.268,159.131
C02453=1026.419,292.813,-128.716,170.647,47.270,159.131
C02454=1026.407,292.398,-128.663,170.639,47.273,159.130
C02455=1026.396,291.982,-128.609,170.631,47.275,159.129
C02456=1026.385,291.566,-128.555,170.625,47.278,159.129
C02457=1026.378,291.318,-128.524,170.620,47.279,159.129
C02458=1026.371,291.070,-128.492,170.614,47.280,159.128
C02459=1026.365,290.823,-128.460,170.611,47.282,159.128
C02460=1026.358,290.574,-128.428,170.606,47.283,159.128
C02461=1026.351,290.326,-128.396,170.602,47.285,159.128
C02462=1026.344,290.078,-128.365,170.597,47.287,159.128
C02463=1026.337,289.831,-128.333,170.593,47.288,159.127
C02464=1026.330,289.583,-128.301,170.588,47.289,159.127
C02465=1026.324,289.335,-128.269,170.584,47.291,159.127
C02466=1026.318,289.087,-128.238,170.579,47.292,159.127
C02467=1026.311,288.839,-128.206,170.574,47.294,159.126
C02468=1026.304,288.591,-128.175,170.570,47.295,159.126
C02469=1026.297,288.344,-128.143,170.565,47.297,159.126
C02470=1026.291,288.096,-128.111,170.561,47.298,159.126
C02471=1026.284,287.848,-128.080,170.556,47.300,159.125
C02472=1026.277,287.600,-128.049,170.552,47.301,159.125
C02473=1026.271,287.352,-128.017,170.548,47.303,159.125
C02474=1026.264,287.104,-127.985,170.544,47.304,159.125
C02475=1026.258,286.856,-127.954,170.539,47.306,159.125
C02476=1026.251,286.608,-127.922,170.535,47.307,159.124
C02477=1026.244,286.360,-127.891,170.530,47.309,159.124
C02478=1026.237,286.113,-127.859,170.526,47.310,159.124
C02479=1026.231,285.865,-127.828,170.521,47.312,159.124
C02480=1026.224,285.617,-127.797,170.516,47.314,159.123
C02481=1026.217,285.369,-127.765,170.513,47.316,159.123
C02482=1026.211,285.121,-127.734,170.508,47.317,159.123
C02483=1026.204,284.873,-127.702,170.504,47.319,159.123
C02484=1026.197,284.625,-127.671,170.499,47.321,159.123
C02485=1026.190,284.377,-127.641,170.495,47.322,159.122
C02486=1026.184,284.130,-127.610,170.490,47.324,159.122
C02487=1026.177,283.882,-127.578,170.487,47.326,159.122
C02488=1026.170,283.634,-127.547,170.482,47.327,159.122
C02489=1026.164,283.385,-127.516,170.478,47.329,159.122
C02490=1026.157,283.138,-127.485,170.473,47.331,159.122
C02491=1026.151,282.890,-127.453,170.469,47.332,159.121
C02492=1026.143,282.642,-127.422,170.464,47.334,159.121
C02493=1026.137,282.393,-127.392,170.461,47.336,159.121
C02494=1026.130,282.146,-127.360,170.456,47.337,159.121
C02495=1026.123,281.898,-127.329,170.452,47.339,159.121
C02496=1026.117,281.650,-127.298,170.447,47.341,159.120
C02497=1026.111,281.402,-127.267,170.443,47.343,159.120
C02498=1026.104,281.154,-127.236,170.438,47.344,159.120
C02499=1026.097,280.906,-127.205,170.435,47.346,159.120
C02500=1026.090,280.658,-127.174,170.430,47.348,159.120
C02501=1026.083,280.410,-127.143,170.426,47.349,159.120
C02502=1026.077,280.162,-127.112,170.421,47.352,159.120
C02503=1026.071,279.914,-127.081,170.417,47.353,159.119
C02504=1026.064,279.666,-127.050,170.413,47.355,159.119
C02505=1026.058,279.418,-127.019,170.409,47.356,159.119
C02506=1026.051,279.170,-126.989,170.404,47.358,159.119
C02507=1026.044,278.922,-126.957,170.400,47.360,159.119
C02508=1026.038,278.674,-126.927,170.395,47.362,159.118
C02509=1026.028,278.270,-126.876,170.389,47.365,159.118
C02510=1026.017,277.867,-126.826,170.382,47.367,159.118
C02511=1026.007,277.463,-126.776,170.375,47.371,159.118
C02512=1025.996,277.060,-126.726,170.368,47.373,159.118
C02513=1025.988,276.812,-126.695,170.364,47.375,159.117
C02514=1025.982,276.564,-126.664,170.360,47.377,159.117
C02515=1025.975,276.315,-126.633,170.356,47.379,159.117
C02516=1025.969,276.068,-126.604,170.351,47.381,159.117
C02517=1025.962,275.819,-126.573,170.347,47.383,159.117
C02518=1025.955,275.571,-126.542,170.343,47.385,159.117
C02519=1025.949,275.324,-126.512,170.339,47.387,159.117
C02520=1025.943,275.075,-126.481,170.334,47.389,159.117
C02521=1025.935,274.827,-126.451,170.331,47.391,159.117
C02522=1025.929,274.579,-126.419,170.326,47.393,159.116
C02523=1025.922,274.332,-126.390,170.322,47.395,159.116
C02524=1025.916,274.083,-126.359,170.319,47.397,159.116
C02525=1025.910,273.835,-126.329,170.314,47.399,159.116
C02526=1025.903,273.587,-126.298,170.310,47.400,159.116
C02527=1025.896,273.338,-126.268,170.305,47.402,159.116
C02528=1025.890,273.092,-126.237,170.302,47.404,159.116
C02529=1025.883,272.843,-126.207,170.297,47.406,159.116
C02530=1025.876,272.595,-126.176,170.293,47.409,159.116
C02531=1025.870,272.347,-126.146,170.289,47.411,159.115
C02532=1025.863,272.099,-126.116,170.285,47.412,159.115
C02533=1025.857,271.851,-126.086,170.281,47.414,159.115
C02534=1025.850,271.603,-126.055,170.277,47.416,159.115
C02535=1025.844,271.354,-126.025,170.273,47.419,159.115
C02536=1025.837,271.107,-125.995,170.268,47.421,159.115
C02537=1025.831,270.858,-125.964,170.265,47.422,159.115
C02538=1025.824,270.611,-125.935,170.260,47.424,159.115
C02539=1025.818,270.362,-125.904,170.256,47.427,159.115
C02540=1025.811,270.115,-125.874,170.252,47.429,159.115
C02541=1025.805,269.866,-125.843,170.248,47.431,159.115
C02542=1025.797,269.618,-125.813,170.244,47.432,159.114
C02543=1025.791,269.370,-125.784,170.240,47.435,159.114
C02544=1025.785,269.121,-125.753,170.236,47.437,159.114
C02545=1025.778,268.874,-125.724,170.231,47.439,159.114
C02546=1025.771,268.626,-125.694,170.228,47.441,159.114
C02547=1025.765,268.378,-125.663,170.223,47.443,159.114
C02548=1025.758,268.129,-125.633,170.220,47.446,159.114
C02549=1025.752,267.881,-125.604,170.216,47.447,159.114
C02550=1025.745,267.633,-125.573,170.211,47.450,159.114
C02551=1025.739,267.385,-125.544,170.208,47.452,159.114
C02552=1025.732,267.137,-125.513,170.203,47.454,159.114
C02553=1025.726,266.889,-125.484,170.200,47.456,159.114
C02554=1025.719,266.640,-125.454,170.195,47.458,159.114
C02555=1025.713,266.393,-125.424,170.191,47.460,159.114
C02556=1025.705,266.145,-125.394,170.188,47.463,159.114
C02557=1025.700,265.896,-125.364,170.183,47.465,159.114
C02558=1025.693,265.648,-125.334,170.180,47.467,159.114
C02559=1025.686,265.400,-125.305,170.175,47.469,159.114
C02560=1025.680,265.152,-125.275,170.172,47.471,159.114
C02561=1025.673,264.904,-125.245,170.167,47.474,159.113
C02562=1025.667,264.656,-125.216,170.163,47.476,159.114
C02563=1025.660,264.408,-125.185,170.160,47.478,159.113
C02564=1025.654,264.159,-125.156,170.155,47.480,159.113
C02565=1025.643,263.760,-125.108,170.149,47.484,159.113
C02566=1025.632,263.361,-125.061,170.143,47.488,159.113
C02567=1025.622,262.962,-125.013,170.137,47.491,159.113
C02568=1025.612,262.564,-124.966,170.130,47.495,159.113
C02569=1025.604,262.315,-124.936,170.126,47.497,159.113
C02570=1025.599,262.067,-124.906,170.122,47.500,159.113
C02571=1025.593,261.819,-124.877,170.119,47.502,159.113
C02572=1025.586,261.571,-124.847,170.114,47.504,159.113
C02573=1025.579,261.323,-124.818,170.110,47.506,159.113
C02574=1025.573,261.075,-124.788,170.106,47.509,159.113
C02575=1025.566,260.826,-124.759,170.103,47.511,159.113
C02576=1025.560,260.578,-124.730,170.099,47.513,159.113
C02577=1025.552,260.330,-124.700,170.094,47.516,159.113
C02578=1025.546,260.082,-124.670,170.091,47.518,159.113
C02579=1025.540,259.834,-124.641,170.087,47.521,159.113
C02580=1025.532,259.585,-124.613,170.083,47.523,159.113
C02581=1025.526,259.337,-124.584,170.079,47.526,159.113
C02582=1025.520,259.089,-124.555,170.075,47.528,159.113
C02583=1025.513,258.841,-124.524,170.072,47.530,159.113
C02584=1025.506,258.593,-124.496,170.067,47.533,159.113
C02585=1025.499,258.345,-124.467,170.064,47.535,159.113
C02586=1025.493,258.096,-124.438,170.059,47.538,159.113
C02587=1025.486,257.848,-124.408,170.056,47.540,159.114
C02588=1025.479,257.600,-124.380,170.052,47.543,159.114
C02589=1025.473,257.351,-124.351,170.048,47.545,159.114
C02590=1025.466,257.103,-124.322,170.044,47.548,159.114
C02591=1025.460,256.855,-124.293,170.040,47.550,159.114
C02592=1025.452,256.606,-124.264,170.037,47.553,159.114
C02593=1025.446,256.358,-124.235,170.032,47.555,159.114
C02594=1025.440,256.110,-124.206,170.029,47.558,159.114
C02595=1025.434,255.862,-124.177,170.025,47.561,159.114
C02596=1025.426,255.613,-124.148,170.021,47.563,159.114
C02597=1025.420,255.365,-124.119,170.018,47.565,159.114
C02598=1025.414,255.117,-124.090,170.013,47.568,159.114
C02599=1025.407,254.869,-124.061,170.010,47.571,159.114
C02600=1025.400,254.620,-124.032,170.006,47.573,159.114
C02601=1025.394,254.372,-124.003,170.002,47.576,159.114
C02602=1025.387,254.124,-123.974,169.999,47.578,159.114
C02603=1025.381,253.876,-123.945,169.994,47.581,159.114
C02604=1025.374,253.628,-123.916,169.991,47.583,159.114
C02605=1025.367,253.379,-123.887,169.986,47.586,159.114
C02606=1025.361,253.131,-123.858,169.983,47.588,159.114
C02607=1025.355,252.883,-123.829,169.980,47.591,159.114
C02608=1025.348,252.635,-123.800,169.975,47.593,159.115
C02609=1025.342,252.386,-123.772,169.972,47.596,159.115
C02610=1025.335,252.138,-123.743,169.967,47.599,159.115
C02611=1025.329,251.890,-123.714,169.964,47.601,159.115
C02612=1025.322,251.642,-123.685,169.961,47.603,159.115
C02613=1025.315,251.394,-123.656,169.956,47.606,159.115
C02614=1025.309,251.145,-123.628,169.953,47.609,159.115
C02615=1025.302,250.897,-123.599,169.949,47.611,159.115
C02616=1025.296,250.649,-123.570,169.945,47.614,159.115
C02617=1025.290,250.401,-123.541,169.942,47.617,159.115
C02618=1025.283,250.152,-123.512,169.937,47.619,159.115
C02619=1025.276,249.903,-123.484,169.934,47.622,159.115
C02620=1025.270,249.655,-123.455,169.931,47.624,159.115
C02621=1025.260,249.255,-123.409,169.925,47.629,159.116
C02622=1025.250,248.855,-123.362,169.919,47.633,159.116
C02623=1025.240,248.454,-123.316,169.913,47.637,159.116
C02624=1025.228,248.053,-123.270,169.907,47.641,159.116
C02625=1025.223,247.805,-123.242,169.902,47.644,159.116
C02626=1025.216,247.557,-123.213,169.899,47.647,159.116
C02627=1025.210,247.308,-123.184,169.896,47.649,159.116
C02628=1025.203,247.060,-123.156,169.891,47.652,159.116
C02629=1025.197,246.812,-123.127,169.888,47.655,159.116
C02630=1025.191,246.564,-123.098,169.885,47.657,159.116
C02631=1025.184,246.315,-123.070,169.880,47.660,159.116
C02632=1025.178,246.067,-123.041,169.877,47.663,159.117
C02633=1025.172,245.818,-123.013,169.874,47.665,159.117
C02634=1025.166,245.570,-122.984,169.869,47.668,159.117
C02635=1025.159,245.322,-122.956,169.866,47.671,159.117
C02636=1025.153,245.074,-122.927,169.863,47.673,159.117
C02637=1025.147,244.826,-122.898,169.858,47.676,159.117
C02638=1025.140,244.577,-122.870,169.855,47.679,159.117
C02639=1025.134,244.329,-122.841,169.852,47.682,159.117
C02640=1025.128,244.081,-122.813,169.847,47.684,159.117
C02641=1025.122,243.833,-122.784,169.844,47.687,159.117
C02642=1025.115,243.584,-122.756,169.841,47.690,159.118
C02643=1025.109,243.336,-122.729,169.836,47.693,159.118
C02644=1025.102,243.088,-122.700,169.833,47.696,159.118
C02645=1025.096,242.839,-122.672,169.830,47.698,159.118
C02646=1025.090,242.591,-122.644,169.825,47.701,159.118
C02647=1025.083,242.343,-122.615,169.822,47.704,159.118
C02648=1025.077,242.094,-122.587,169.819,47.706,159.118
C02649=1025.070,241.846,-122.559,169.815,47.710,159.118
C02650=1025.063,241.598,-122.531,169.811,47.712,159.119
C02651=1025.057,241.349,-122.502,169.808,47.715,159.119
C02652=1025.051,241.101,-122.475,169.804,47.718,159.119
C02653=1025.045,240.852,-122.446,169.801,47.721,159.119
C02654=1025.038,240.605,-122.418,169.797,47.723,159.119
C02655=1025.032,240.356,-122.390,169.793,47.727,159.119
C02656=1025.026,240.107,-122.362,169.790,47.729,159.119
C02657=1025.019,239.859,-122.334,169.787,47.732,159.120
C02658=1025.013,239.610,-122.306,169.782,47.735,159.120
C02659=1025.006,239.362,-122.278,169.779,47.738,159.120
C02660=1024.999,239.114,-122.250,169.775,47.742,159.120
C02661=1024.993,238.866,-122.222,169.772,47.744,159.120
C02662=1024.986,238.617,-122.194,169.769,47.747,159.120
C02663=1024.980,238.369,-122.167,169.765,47.750,159.121
C02664=1024.974,238.121,-122.139,169.761,47.753,159.121
C02665=1024.967,237.872,-122.111,169.758,47.756,159.121
C02666=1024.961,237.624,-122.083,169.754,47.759,159.121
C02667=1024.954,237.375,-122.056,169.751,47.762,159.121
C02668=1024.947,237.127,-122.028,169.747,47.765,159.121
C02669=1024.941,236.878,-122.000,169.743,47.768,159.122
C02670=1024.935,236.630,-121.972,169.740,47.771,159.122
C02671=1024.929,236.382,-121.944,169.736,47.774,159.122
C02672=1024.922,236.133,-121.917,169.733,47.777,159.122
C02673=1024.915,235.885,-121.889,169.730,47.780,159.122
C02674=1024.908,235.637,-121.861,169.725,47.783,159.122
C02675=1024.902,235.388,-121.834,169.722,47.786,159.123
C02676=1024.896,235.140,-121.806,169.718,47.789,159.123
C02677=1024.885,234.733,-121.761,169.713,47.795,159.123
C02678=1024.875,234.326,-121.716,169.707,47.799,159.123
C02679=1024.864,233.919,-121.670,169.701,47.805,159.124
C02680=1024.853,233.513,-121.626,169.696,47.809,159.124
C02681=1024.847,233.264,-121.598,169.692,47.812,159.124
C02682=1024.841,233.016,-121.569,169.688,47.816,159.124
C02683=1024.835,232.767,-121.543,169.685,47.819,159.125
C02684=1024.828,232.519,-121.515,169.682,47.822,159.125
C02685=1024.822,232.270,-121.487,169.678,47.825,159.125
C02686=1024.815,232.022,-121.460,169.675,47.828,159.125
C02687=1024.809,231.774,-121.432,169.671,47.831,159.125
C02688=1024.802,231.525,-121.405,169.668,47.834,159.126
C02689=1024.796,231.277,-121.378,169.664,47.837,159.126
C02690=1024.790,231.029,-121.350,169.660,47.841,159.126
C02691=1024.783,230.781,-121.322,169.657,47.844,159.126
C02692=1024.777,230.532,-121.295,169.654,47.847,159.126
C02693=1024.770,230.283,-121.268,169.650,47.850,159.127
C02694=1024.764,230.035,-121.240,169.647,47.853,159.127
C02695=1024.757,229.786,-121.213,169.644,47.856,159.127
C02696=1024.751,229.538,-121.186,169.639,47.859,159.127
C02697=1024.745,229.290,-121.158,169.636,47.862,159.127
C02698=1024.738,229.041,-121.131,169.633,47.865,159.128
C02699=1024.732,228.793,-121.103,169.629,47.869,159.128
C02700=1024.726,228.544,-121.077,169.626,47.872,159.128
C02701=1024.719,228.296,-121.049,169.623,47.875,159.128
C02702=1024.713,228.047,-121.022,169.619,47.878,159.128
C02703=1024.707,227.799,-120.995,169.616,47.881,159.129
C02704=1024.699,227.551,-120.968,169.613,47.885,159.129
C02705=1024.693,227.302,-120.941,169.609,47.889,159.129
C02706=1024.687,227.054,-120.913,169.606,47.892,159.130
C02707=1024.681,226.805,-120.886,169.602,47.895,159.130
C02708=1024.674,226.557,-120.858,169.599,47.898,159.130
C02709=1024.667,226.309,-120.832,169.596,47.901,159.130
C02710=1024.661,226.059,-120.805,169.592,47.905,159.130
C02711=1024.654,225.811,-120.778,169.589,47.908,159.131
C02712=1024.648,225.563,-120.752,169.585,47.912,159.131
C02713=1024.641,225.315,-120.724,169.582,47.915,159.131
C02714=1024.635,225.066,-120.697,169.579,47.918,159.131
C02715=1024.628,224.817,-120.671,169.574,47.921,159.132
C02716=1024.622,224.569,-120.643,169.571,47.925,159.132
C02717=1024.616,224.321,-120.616,169.569,47.928,159.132
C02718=1024.609,224.072,-120.590,169.565,47.932,159.132
C02719=1024.603,223.824,-120.563,169.561,47.935,159.133
C02720=1024.596,223.575,-120.536,169.557,47.938,159.133
C02721=1024.589,223.326,-120.509,169.554,47.941,159.133
C02722=1024.583,223.078,-120.483,169.552,47.945,159.134
C02723=1024.577,222.830,-120.455,169.547,47.948,159.134
C02724=1024.571,222.581,-120.428,169.544,47.952,159.134
C02725=1024.564,222.332,-120.402,169.541,47.955,159.134
C02726=1024.558,222.085,-120.374,169.538,47.959,159.135
C02727=1024.551,221.836,-120.347,169.534,47.962,159.135
C02728=1024.544,221.587,-120.321,169.531,47.965,159.135
C02729=1024.538,221.339,-120.294,169.527,47.968,159.135
C02730=1024.532,221.090,-120.267,169.525,47.972,159.136
C02731=1024.525,220.842,-120.241,169.520,47.976,159.136
C02732=1024.519,220.593,-120.214,169.517,47.979,159.136
C02733=1024.508,220.178,-120.169,169.512,47.985,159.137
C02734=1024.498,219.764,-120.125,169.507,47.990,159.137
C02735=1024.487,219.349,-120.080,169.501,47.996,159.138
C02736=1024.476,218.935,-120.035,169.495,48.002,159.138
C02737=1024.470,218.686,-120.009,169.492,48.005,159.138
C02738=1024.463,218.438,-119.982,169.488,48.009,159.139
C02739=1024.458,218.189,-119.956,169.486,48.012,159.139
C02740=1024.450,217.941,-119.929,169.481,48.016,159.139
C02741=1024.444,217.693,-119.903,169.479,48.020,159.140
C02742=1024.438,217.443,-119.876,169.476,48.023,159.140
C02743=1024.431,217.195,-119.850,169.472,48.027,159.140
C02744=1024.425,216.946,-119.823,169.469,48.030,159.140
C02745=1024.418,216.698,-119.797,169.465,48.034,159.141
C02746=1024.411,216.450,-119.771,169.462,48.037,159.141
C02747=1024.405,216.201,-119.744,169.459,48.041,159.141
C02748=1024.398,215.952,-119.718,169.455,48.044,159.142
C02749=1024.392,215.704,-119.692,169.452,48.048,159.142
C02750=1024.385,215.455,-119.665,169.448,48.052,159.142
C02751=1024.379,215.207,-119.639,169.446,48.055,159.143
C02752=1024.373,214.959,-119.612,169.443,48.059,159.143
C02753=1024.366,214.710,-119.585,169.439,48.062,159.143
C02754=1024.360,214.462,-119.560,169.436,48.066,159.144
C02755=1024.353,214.212,-119.533,169.433,48.069,159.144
C02756=1024.347,213.964,-119.507,169.429,48.073,159.144
C02757=1024.340,213.716,-119.481,169.426,48.077,159.144
C02758=1024.334,213.467,-119.454,169.422,48.081,159.145
C02759=1024.327,213.219,-119.428,169.420,48.084,159.145
C02760=1024.321,212.970,-119.401,169.416,48.088,159.145
C02761=1024.315,212.722,-119.376,169.413,48.092,159.146
C02762=1024.308,212.473,-119.350,169.410,48.095,159.146
C02763=1024.302,212.224,-119.323,169.406,48.099,159.146
C02764=1024.295,211.976,-119.296,169.403,48.103,159.147
C02765=1024.288,211.728,-119.270,169.400,48.106,159.147
C02766=1024.283,211.479,-119.244,169.396,48.110,159.147
C02767=1024.276,211.231,-119.218,169.394,48.114,159.148
C02768=1024.270,210.981,-119.191,169.390,48.117,159.148
C02769=1024.263,210.733,-119.165,169.387,48.121,159.148
C02770=1024.257,210.485,-119.140,169.384,48.125,159.149
C02771=1024.251,210.236,-119.113,169.381,48.128,159.149
C02772=1024.244,209.988,-119.087,169.377,48.132,159.149
C02773=1024.238,209.739,-119.061,169.374,48.136,159.150
C02774=1024.231,209.490,-119.035,169.371,48.140,159.150
C02775=1024.224,209.242,-119.009,169.368,48.143,159.150
C02776=1024.218,208.994,-118.983,169.364,48.147,159.151
C02777=1024.212,208.744,-118.956,169.361,48.151,159.151
C02778=1024.206,208.496,-118.931,169.358,48.155,159.152
C02779=1024.199,208.248,-118.905,169.354,48.158,159.152
C02780=1024.193,208.000,-118.879,169.352,48.162,159.152
C02781=1024.186,207.750,-118.853,169.348,48.166,159.153
C02782=1024.179,207.502,-118.827,169.345,48.170,159.153
C02783=1024.173,207.254,-118.802,169.342,48.173,159.153
C02784=1024.167,207.005,-118.775,169.339,48.178,159.154
C02785=1024.161,206.756,-118.750,169.335,48.181,159.154
C02786=1024.154,206.508,-118.723,169.332,48.185,159.154
C02787=1024.148,206.259,-118.698,169.329,48.189,159.155
C02788=1024.141,206.010,-118.672,169.326,48.192,159.155
C02789=1024.131,205.598,-118.629,169.320,48.199,159.156
C02790=1024.119,205.186,-118.587,169.315,48.205,159.156
C02791=1024.108,204.775,-118.544,169.311,48.212,159.157
C02792=1024.098,204.363,-118.501,169.304,48.218,159.158
C02793=1024.074,203.330,-118.401,168.894,48.119,159.079
C02794=1024.068,203.082,-118.376,168.891,48.124,159.080
C02795=1024.063,202.833,-118.352,168.886,48.128,159.080
C02796=1024.057,202.584,-118.328,168.882,48.133,159.080
C02797=1024.051,202.336,-118.304,168.878,48.138,159.081
C02798=1024.046,202.087,-118.279,168.873,48.142,159.081
C02799=1024.041,201.838,-118.256,168.870,48.147,159.082
C02800=1024.034,201.589,-118.232,168.865,48.152,159.082
C02801=1024.029,201.340,-118.208,168.862,48.157,159.083
C02802=1024.024,201.092,-118.183,168.857,48.161,159.083
C02803=1024.018,200.843,-118.159,168.854,48.166,159.083
C02804=1024.012,200.594,-118.135,168.849,48.171,159.084
C02805=1024.007,200.346,-118.111,168.846,48.176,159.084
C02806=1024.001,200.097,-118.087,168.841,48.180,159.084
C02807=1023.996,199.847,-118.063,168.836,48.185,159.085
C02808=1023.990,199.599,-118.039,168.833,48.190,159.085
C02809=1023.984,199.350,-118.015,168.828,48.195,159.086
C02810=1023.978,199.101,-117.991,168.825,48.200,159.086
C02811=1023.972,198.852,-117.968,168.820,48.205,159.087
C02812=1023.967,198.604,-117.944,168.816,48.210,159.087
C02813=1023.961,198.356,-117.920,168.813,48.215,159.088
C02814=1023.955,198.106,-117.896,168.808,48.220,159.088
C02815=1023.949,197.857,-117.872,168.805,48.225,159.089
C02816=1023.943,197.608,-117.849,168.800,48.230,159.089
C02817=1023.938,197.360,-117.825,168.796,48.234,159.089
C02818=1023.931,197.111,-117.801,168.792,48.239,159.090
C02819=1023.926,196.862,-117.778,168.787,48.244,159.090
C02820=1023.920,196.613,-117.754,168.784,48.249,159.091
C02821=1023.915,196.365,-117.731,168.780,48.254,159.091
C02822=1023.909,196.116,-117.707,168.776,48.259,159.091
C02823=1023.903,195.866,-117.683,168.772,48.264,159.092
C02824=1023.898,195.618,-117.659,168.768,48.268,159.092
C02825=1023.892,195.369,-117.636,168.764,48.274,159.093
C02826=1023.886,195.121,-117.612,168.760,48.278,159.093
C02827=1023.881,194.871,-117.589,168.756,48.283,159.094
C02828=1023.875,194.623,-117.565,168.751,48.288,159.094
C02829=1023.868,194.373,-117.542,168.748,48.293,159.095
C02830=1023.863,194.125,-117.518,168.743,48.298,159.095
C02831=1023.857,193.876,-117.495,168.740,48.303,159.096
C02832=1023.852,193.627,-117.471,168.736,48.308,159.096
C02833=1023.846,193.379,-117.448,168.732,48.313,159.096
C02834=1023.840,193.130,-117.424,168.728,48.318,159.097
C02835=1023.835,192.881,-117.400,168.724,48.323,159.097
C02836=1023.830,192.632,-117.377,168.720,48.328,159.098
C02837=1023.824,192.384,-117.353,168.716,48.333,159.098
C02838=1023.819,192.135,-117.330,168.713,48.338,159.099
C02839=1023.812,191.886,-117.306,168.708,48.343,159.099
C02840=1023.807,191.636,-117.283,168.705,48.347,159.100
C02841=1023.801,191.388,-117.260,168.701,48.353,159.100
C02842=1023.795,191.139,-117.236,168.697,48.357,159.101
C02843=1023.790,190.890,-117.213,168.693,48.362,159.101
C02844=1023.784,190.641,-117.190,168.689,48.367,159.101
C02845=1023.778,190.393,-117.166,168.685,48.372,159.102
C02846=1023.773,190.144,-117.142,168.681,48.377,159.102
C02847=1023.768,189.895,-117.119,168.677,48.382,159.103
C02848=1023.762,189.646,-117.095,168.673,48.387,159.103
C02849=1023.757,189.397,-117.072,168.670,48.392,159.104
C02850=1023.751,189.148,-117.049,168.666,48.397,159.104
C02851=1023.746,188.899,-117.026,168.662,48.402,159.105
C02852=1023.740,188.651,-117.002,168.658,48.407,159.105
C02853=1023.734,188.402,-116.979,168.654,48.412,159.106
C02854=1023.729,188.120,-116.952,168.650,48.417,159.106
C02855=1023.722,187.837,-116.926,168.646,48.423,159.107
C02856=1023.716,187.555,-116.900,168.642,48.428,159.107
C02857=1023.709,187.273,-116.873,168.636,48.434,159.108
C02858=1023.704,187.024,-116.850,168.633,48.439,159.108
C02859=1023.699,186.775,-116.827,168.630,48.444,159.109
C02860=1023.693,186.526,-116.804,168.625,48.449,159.109
C02861=1023.688,186.277,-116.780,168.622,48.454,159.110
C02862=1023.682,186.029,-116.757,168.618,48.459,159.110
C02863=1023.676,185.780,-116.734,168.614,48.464,159.110
C02864=1023.671,185.531,-116.710,168.610,48.469,159.111
C02865=1023.666,185.283,-116.688,168.607,48.473,159.111
C02866=1023.660,185.034,-116.665,168.602,48.479,159.112
C02867=1023.655,184.784,-116.641,168.599,48.484,159.113
C02868=1023.650,184.536,-116.618,168.596,48.489,159.113
C02869=1023.644,184.287,-116.595,168.592,48.494,159.113
C02870=1023.639,184.037,-116.572,168.588,48.499,159.114
C02871=1023.633,183.789,-116.549,168.585,48.504,159.114
C02872=1023.627,183.540,-116.525,168.580,48.509,159.115
C02873=1023.623,183.292,-116.502,168.577,48.514,159.115
C02874=1023.617,183.043,-116.479,168.573,48.518,159.116
C02875=1023.612,182.793,-116.457,168.569,48.523,159.116
C02876=1023.607,182.544,-116.433,168.566,48.528,159.117
C02877=1023.601,182.295,-116.410,168.562,48.533,159.117
C02878=1023.595,182.046,-116.387,168.558,48.539,159.118
C02879=1023.589,181.798,-116.365,168.555,48.544,159.118
C02880=1023.583,181.548,-116.343,168.550,48.549,159.119
C02881=1023.578,181.299,-116.320,168.547,48.554,159.119
C02882=1023.572,181.050,-116.297,168.543,48.559,159.120
C02883=1023.566,180.803,-116.275,168.539,48.564,159.120
C02884=1023.561,180.553,-116.253,168.536,48.570,159.121
C02885=1023.555,180.304,-116.230,168.532,48.575,159.121
C02886=1023.548,180.056,-116.207,168.529,48.580,159.122
C02887=1023.543,179.806,-116.185,168.524,48.586,159.122
C02888=1023.537,179.557,-116.162,168.521,48.590,159.123
C02889=1023.531,179.308,-116.139,168.518,48.596,159.123
C02890=1023.526,179.060,-116.118,168.513,48.601,159.124
C02891=1023.520,178.811,-116.095,168.510,48.607,159.125
C02892=1023.515,178.561,-116.073,168.506,48.612,159.125
C02893=1023.508,178.313,-116.050,168.502,48.616,159.125
C02894=1023.503,178.064,-116.028,168.499,48.622,159.126
C02895=1023.497,177.814,-116.005,168.495,48.627,159.127
C02896=1023.492,177.566,-115.983,168.492,48.633,159.127
C02897=1023.486,177.317,-115.961,168.488,48.638,159.128
C02898=1023.480,177.068,-115.938,168.484,48.643,159.128
C02899=1023.474,176.819,-115.915,168.481,48.648,159.129
C02900=1023.468,176.570,-115.894,168.476,48.653,159.129
C02901=1023.463,176.322,-115.871,168.473,48.659,159.130
C02902=1023.458,176.072,-115.849,168.470,48.664,159.130
C02903=1023.452,175.823,-115.826,168.465,48.669,159.131
C02904=1023.446,175.574,-115.804,168.462,48.674,159.131
C02905=1023.441,175.326,-115.782,168.459,48.679,159.132
C02906=1023.435,175.076,-115.759,168.455,48.685,159.132
C02907=1023.429,174.828,-115.737,168.451,48.690,159.133
C02908=1023.423,174.578,-115.715,168.448,48.695,159.133
C02909=1023.418,174.330,-115.692,168.444,48.700,159.134
C02910=1023.412,174.081,-115.671,168.441,48.705,159.134
C02911=1023.407,173.831,-115.648,168.438,48.711,159.135
C02912=1023.401,173.583,-115.626,168.434,48.716,159.136
C02913=1023.396,173.334,-115.603,168.430,48.721,159.136
C02914=1023.390,173.085,-115.581,168.427,48.726,159.137
C02915=1023.385,172.836,-115.559,168.423,48.731,159.137
C02916=1023.379,172.587,-115.537,168.419,48.737,159.138
C02917=1023.373,172.338,-115.515,168.416,48.742,159.138
C02918=1023.367,172.055,-115.490,168.412,48.748,159.139
C02919=1023.360,171.773,-115.465,168.408,48.754,159.139
C02920=1023.354,171.491,-115.439,168.403,48.759,159.140
C02921=1023.348,171.207,-115.414,168.400,48.766,159.141
C02922=1023.342,170.959,-115.392,168.396,48.771,159.141
C02923=1023.337,170.710,-115.369,168.393,48.776,159.142
C02924=1023.332,170.461,-115.348,168.389,48.781,159.142
C02925=1023.326,170.212,-115.325,168.385,48.786,159.143
C02926=1023.320,169.963,-115.303,168.382,48.792,159.143
C02927=1023.315,169.714,-115.281,168.379,48.797,159.144
C02928=1023.309,169.465,-115.260,168.375,48.802,159.144
C02929=1023.303,169.216,-115.237,168.372,48.807,159.145
C02930=1023.299,168.967,-115.215,168.368,48.812,159.145
C02931=1023.292,168.718,-115.193,168.365,48.818,159.146
C02932=1023.287,168.469,-115.171,168.362,48.823,159.147
C02933=1023.282,168.220,-115.148,168.358,48.829,159.147
C02934=1023.276,167.971,-115.127,168.354,48.833,159.148
C02935=1023.271,167.722,-115.105,168.351,48.838,159.148
C02936=1023.265,167.472,-115.083,168.348,48.844,159.149
C02937=1023.260,167.225,-115.061,168.344,48.849,159.149
C02938=1023.254,166.975,-115.038,168.340,48.855,159.150
C02939=1023.249,166.726,-115.016,168.337,48.859,159.150
C02940=1023.243,166.477,-114.995,168.334,48.864,159.151
C02941=1023.238,166.228,-114.973,168.330,48.870,159.151
C02942=1023.233,165.979,-114.950,168.327,48.875,159.152
C02943=1023.227,165.731,-114.929,168.324,48.880,159.153
C02944=1023.222,165.481,-114.907,168.320,48.885,159.153
C02945=1023.217,165.232,-114.885,168.316,48.890,159.153
C02946=1023.211,164.983,-114.863,168.313,48.896,159.154
C02947=1023.206,164.734,-114.841,168.310,48.901,159.155
C02948=1023.200,164.485,-114.819,168.307,48.906,159.155
C02949=1023.195,164.237,-114.797,168.303,48.911,159.156
C02950=1023.189,163.987,-114.775,168.299,48.916,159.156
C02951=1023.184,163.739,-114.753,168.296,48.922,159.157
C02952=1023.178,163.489,-114.731,168.293,48.927,159.157
C02953=1023.173,163.241,-114.709,168.289,48.932,159.158
C02954=1023.168,162.991,-114.687,168.286,48.937,159.158
C02955=1023.162,162.743,-114.666,168.283,48.942,159.159
C02956=1023.157,162.494,-114.644,168.280,48.948,159.160
C02957=1023.152,162.244,-114.622,168.276,48.953,159.160
C02958=1023.146,161.996,-114.601,168.273,48.958,159.161
C02959=1023.141,161.746,-114.578,168.269,48.963,159.161
C02960=1023.136,161.497,-114.556,168.265,48.968,159.162
C02961=1023.130,161.248,-114.535,168.262,48.974,159.162
C02962=1023.125,160.999,-114.513,168.259,48.979,159.163
C02963=1023.120,160.751,-114.492,168.256,48.984,159.163
C02964=1023.114,160.501,-114.469,168.253,48.989,159.164
C02965=1023.109,160.253,-114.448,168.249,48.994,159.164
C02966=1023.103,160.003,-114.426,168.246,49.000,159.165
C02967=1023.098,159.755,-114.404,168.243,49.005,159.165
C02968=1023.094,159.506,-114.382,168.240,49.010,159.166
C02969=1023.087,159.257,-114.361,168.236,49.015,159.167
C02970=1023.083,159.008,-114.339,168.233,49.020,159.167
C02971=1023.076,158.759,-114.317,168.229,49.026,159.168
C02972=1023.071,158.509,-114.297,168.226,49.031,159.168
C02973=1023.066,158.261,-114.275,168.223,49.036,159.169
C02974=1023.060,158.011,-114.253,168.220,49.042,159.169
C02975=1023.055,157.763,-114.232,168.217,49.047,159.170
C02976=1023.049,157.513,-114.211,168.213,49.052,159.171
C02977=1023.043,157.265,-114.190,168.209,49.058,159.171
C02978=1023.038,157.016,-114.168,168.206,49.064,159.172
C02979=1023.033,156.766,-114.147,168.203,49.069,159.172
C02980=1023.027,156.517,-114.125,168.200,49.074,159.173
C02981=1023.021,156.269,-114.104,168.196,49.079,159.173
C02982=1023.015,155.985,-114.080,168.193,49.086,159.174
C02983=1023.008,155.702,-114.056,168.189,49.092,159.175
C02984=1023.002,155.419,-114.032,168.185,49.098,159.176
C02985=1022.996,155.136,-114.008,168.181,49.104,159.176
C02986=1022.991,154.887,-113.986,168.178,49.110,159.177
C02987=1022.986,154.638,-113.965,168.174,49.115,159.177
C02988=1022.980,154.389,-113.944,168.171,49.120,159.178
C02989=1022.974,154.140,-113.923,168.168,49.125,159.178
C02990=1022.969,153.891,-113.902,168.165,49.131,159.179
C02991=1022.963,153.642,-113.880,168.162,49.136,159.180
C02992=1022.958,153.393,-113.859,168.159,49.141,159.180
C02993=1022.952,153.144,-113.838,168.156,49.147,159.181
C02994=1022.947,152.894,-113.817,168.153,49.152,159.181
C02995=1022.941,152.646,-113.796,168.148,49.158,159.182
C02996=1022.936,152.397,-113.775,168.145,49.163,159.183
C02997=1022.930,152.148,-113.754,168.142,49.169,159.183
C02998=1022.924,151.898,-113.733,168.139,49.174,159.184
C02999=1022.919,151.650,-113.712,168.136,49.179,159.184
C03000=1022.914,151.401,-113.691,168.133,49.185,159.185
C03001=1022.907,151.152,-113.670,168.129,49.190,159.185
C03002=1022.902,150.902,-113.649,168.126,49.195,159.186
C03003=1022.897,150.654,-113.628,168.123,49.201,159.187
C03004=1022.891,150.404,-113.607,168.119,49.206,159.187
C03005=1022.885,150.155,-113.586,168.116,49.212,159.188
C03006=1022.880,149.906,-113.565,168.113,49.218,159.188
C03007=1022.875,149.657,-113.544,168.110,49.222,159.189
C03008=1022.868,149.408,-113.523,168.107,49.228,159.190
C03009=1022.863,149.159,-113.502,168.104,49.234,159.190
C03010=1022.858,148.910,-113.482,168.100,49.239,159.191
C03011=1022.852,148.661,-113.460,168.097,49.244,159.191
C03012=1022.847,148.412,-113.440,168.094,49.250,159.192
C03013=1022.841,148.162,-113.419,168.091,49.255,159.193
C03014=1022.836,147.914,-113.398,168.088,49.260,159.193
C03015=1022.830,147.665,-113.377,168.085,49.266,159.194
C03016=1022.825,147.416,-113.357,168.082,49.272,159.194
C03017=1022.819,147.167,-113.335,168.079,49.276,159.195
C03018=1022.814,146.917,-113.314,168.076,49.282,159.196
C03019=1022.809,146.668,-113.294,168.071,49.288,159.196
C03020=1022.803,146.419,-113.273,168.068,49.293,159.197
C03021=1022.798,146.171,-113.252,168.065,49.299,159.197
C03022=1022.792,145.921,-113.231,168.062,49.304,159.198
C03023=1022.787,145.672,-113.211,168.059,49.310,159.199
C03024=1022.781,145.423,-113.191,168.056,49.315,159.199
C03025=1022.775,145.174,-113.170,168.053,49.320,159.200
C03026=1022.770,144.925,-113.149,168.050,49.326,159.200
C03027=1022.764,144.675,-113.128,168.047,49.332,159.201
C03028=1022.758,144.427,-113.108,168.044,49.337,159.202
C03029=1022.753,144.177,-113.087,168.040,49.342,159.202
C03030=1022.747,143.928,-113.067,168.037,49.348,159.203
C03031=1022.742,143.679,-113.046,168.034,49.353,159.203
C03032=1022.736,143.430,-113.026,168.031,49.359,159.204
C03033=1022.730,143.181,-113.005,168.027,49.365,159.205
C03034=1022.725,142.932,-112.984,168.024,49.370,159.205
C03035=1022.720,142.683,-112.964,168.021,49.376,159.206
C03036=1022.714,142.434,-112.944,168.018,49.381,159.206
C03037=1022.708,142.185,-112.923,168.015,49.387,159.207
C03038=1022.703,141.936,-112.902,168.012,49.392,159.208
C03039=1022.698,141.687,-112.882,168.009,49.397,159.208
C03040=1022.691,141.437,-112.862,168.006,49.403,159.209
C03041=1022.686,141.188,-112.841,168.003,49.409,159.210
C03042=1022.681,140.939,-112.820,168.000,49.414,159.210
C03043=1022.675,140.690,-112.800,167.997,49.419,159.211
C03044=1022.669,140.441,-112.780,167.994,49.425,159.211
C03045=1022.664,140.192,-112.759,167.991,49.431,159.212
C03046=1022.658,139.909,-112.736,167.987,49.436,159.213
C03047=1022.651,139.626,-112.713,167.984,49.443,159.213
C03048=1022.645,139.342,-112.690,167.980,49.449,159.214
C03049=1022.639,139.058,-112.666,167.976,49.455,159.215
C03050=1022.633,138.809,-112.646,167.973,49.461,159.215
C03051=1022.628,138.560,-112.626,167.970,49.466,159.216
C03052=1022.623,138.311,-112.605,167.967,49.472,159.217
C03053=1022.617,138.062,-112.585,167.964,49.477,159.217
C03054=1022.611,137.813,-112.565,167.961,49.483,159.218
C03055=1022.606,137.564,-112.544,167.958,49.489,159.218
C03056=1022.601,137.315,-112.525,167.955,49.494,159.219
C03057=1022.595,137.066,-112.504,167.952,49.499,159.220
C03058=1022.589,136.817,-112.484,167.949,49.505,159.220
C03059=1022.584,136.568,-112.464,167.946,49.510,159.221
C03060=1022.578,136.319,-112.444,167.943,49.516,159.222
C03061=1022.573,136.070,-112.423,167.940,49.522,159.222
C03062=1022.568,135.820,-112.403,167.937,49.527,159.223
C03063=1022.562,135.571,-112.383,167.934,49.532,159.223
C03064=1022.557,135.322,-112.363,167.931,49.538,159.224
C03065=1022.551,135.073,-112.343,167.928,49.544,159.225
C03066=1022.544,134.824,-112.323,167.925,49.549,159.225
C03067=1022.539,134.574,-112.303,167.922,49.555,159.226
C03068=1022.533,134.325,-112.283,167.918,49.560,159.226
C03069=1022.528,134.076,-112.262,167.915,49.566,159.227
C03070=1022.522,133.827,-112.243,167.912,49.571,159.228
C03071=1022.517,133.577,-112.222,167.909,49.577,159.228
C03072=1022.511,133.329,-112.202,167.906,49.583,159.229
C03073=1022.506,133.080,-112.182,167.904,49.588,159.230
C03074=1022.501,132.831,-112.163,167.901,49.594,159.230
C03075=1022.495,132.582,-112.142,167.897,49.599,159.231
C03076=1022.489,132.333,-112.123,167.894,49.605,159.231
C03077=1022.484,132.083,-112.103,167.891,49.610,159.232
C03078=1022.478,131.834,-112.083,167.888,49.616,159.233
C03079=1022.473,131.585,-112.062,167.885,49.622,159.233
C03080=1022.467,131.336,-112.043,167.882,49.627,159.234
C03081=1022.462,131.087,-112.022,167.879,49.632,159.235
C03082=1022.456,130.838,-112.002,167.876,49.638,159.235
C03083=1022.451,130.588,-111.983,167.874,49.643,159.236
C03084=1022.445,130.339,-111.963,167.871,49.649,159.237
C03085=1022.439,130.090,-111.943,167.868,49.655,159.237
C03086=1022.434,129.841,-111.923,167.865,49.660,159.238
C03087=1022.429,129.591,-111.904,167.862,49.665,159.238
C03088=1022.423,129.342,-111.884,167.859,49.671,159.239
C03089=1022.417,129.093,-111.864,167.856,49.677,159.240
C03090=1022.411,128.844,-111.844,167.852,49.683,159.240
C03091=1022.405,128.595,-111.825,167.849,49.688,159.241
C03092=1022.399,128.346,-111.805,167.846,49.694,159.242
C03093=1022.394,128.096,-111.785,167.843,49.700,159.242
C03094=1022.388,127.847,-111.765,167.840,49.705,159.243
C03095=1022.383,127.599,-111.747,167.837,49.711,159.243
C03096=1022.377,127.349,-111.727,167.834,49.717,159.244
C03097=1022.371,127.100,-111.707,167.831,49.722,159.245
C03098=1022.366,126.851,-111.688,167.829,49.728,159.245
C03099=1022.360,126.602,-111.668,167.826,49.734,159.246
C03100=1022.355,126.352,-111.648,167.823,49.739,159.247
C03101=1022.349,126.103,-111.629,167.820,49.745,159.247
C03102=1022.343,125.854,-111.609,167.817,49.751,159.248
C03103=1022.337,125.605,-111.590,167.814,49.756,159.249
C03104=1022.332,125.355,-111.571,167.811,49.762,159.249
C03105=1022.326,125.107,-111.551,167.808,49.768,159.250
C03106=1022.321,124.858,-111.532,167.805,49.773,159.251
C03107=1022.315,124.608,-111.513,167.802,49.779,159.251
C03108=1022.310,124.359,-111.492,167.799,49.785,159.252
C03109=1022.304,124.110,-111.473,167.797,49.790,159.253
C03110=1022.298,123.826,-111.450,167.794,49.797,159.253
C03111=1022.291,123.544,-111.429,167.790,49.803,159.254
C03112=1022.284,123.260,-111.407,167.787,49.809,159.255
C03113=1022.278,122.977,-111.385,167.783,49.816,159.256
C03114=1022.273,122.728,-111.366,167.780,49.822,159.256
C03115=1022.267,122.478,-111.345,167.778,49.827,159.257
C03116=1022.262,122.229,-111.326,167.774,49.832,159.257
C03117=1022.256,121.980,-111.306,167.771,49.838,159.258
C03118=1022.251,121.731,-111.288,167.768,49.844,159.259
C03119=1022.245,121.482,-111.268,167.765,49.849,159.259
C03120=1022.239,121.233,-111.248,167.763,49.855,159.260
C03121=1022.234,120.983,-111.229,167.760,49.861,159.261
C03122=1022.228,120.734,-111.210,167.758,49.866,159.261
C03123=1022.223,120.485,-111.191,167.755,49.872,159.262
C03124=1022.218,120.236,-111.170,167.752,49.878,159.263
C03125=1022.212,119.986,-111.151,167.749,49.883,159.263
C03126=1022.206,119.737,-111.132,167.746,49.888,159.264
C03127=1022.200,119.488,-111.113,167.743,49.894,159.264
C03128=1022.195,119.239,-111.094,167.740,49.900,159.265
C03129=1022.189,118.990,-111.074,167.737,49.905,159.266
C03130=1022.184,118.741,-111.055,167.734,49.911,159.266
C03131=1022.178,118.491,-111.035,167.731,49.917,159.267
C03132=1022.173,118.242,-111.017,167.728,49.923,159.268
C03133=1022.167,117.993,-110.997,167.726,49.928,159.268
C03134=1022.162,117.743,-110.977,167.723,49.933,159.269
C03135=1022.156,117.494,-110.958,167.720,49.939,159.270
C03136=1022.151,117.246,-110.939,167.717,49.944,159.270
C03137=1022.146,116.996,-110.919,167.714,49.950,159.271
C03138=1022.140,116.747,-110.900,167.711,49.956,159.272
C03139=1022.134,116.497,-110.881,167.708,49.962,159.272
C03140=1022.129,116.249,-110.862,167.705,49.967,159.273
C03141=1022.123,115.999,-110.843,167.703,49.972,159.273
C03142=1022.118,115.750,-110.824,167.700,49.978,159.274
C03143=1022.113,115.501,-110.805,167.697,49.983,159.275
C03144=1022.107,115.252,-110.784,167.694,49.989,159.275
C03145=1022.102,115.002,-110.765,167.691,49.995,159.276
C03146=1022.097,114.754,-110.746,167.688,50.000,159.276
C03147=1022.091,114.504,-110.727,167.685,50.006,159.277
C03148=1022.085,114.255,-110.708,167.683,50.011,159.278
C03149=1022.080,114.006,-110.689,167.680,50.017,159.278
C03150=1022.074,113.757,-110.669,167.677,50.022,159.279
C03151=1022.069,113.507,-110.650,167.675,50.028,159.280
C03152=1022.064,113.259,-110.631,167.671,50.033,159.280
C03153=1022.058,113.009,-110.612,167.668,50.039,159.281
C03154=1022.052,112.760,-110.593,167.666,50.044,159.282
C03155=1022.048,112.511,-110.573,167.664,50.050,159.282
C03156=1022.042,112.262,-110.555,167.661,50.056,159.283
C03157=1022.036,112.012,-110.535,167.658,50.061,159.284
C03158=1022.031,111.763,-110.517,167.655,50.067,159.284
C03159=1022.025,111.513,-110.498,167.652,50.072,159.285
C03160=1022.020,111.264,-110.479,167.649,50.078,159.285
C03161=1022.014,111.015,-110.460,167.646,50.084,159.286
C03162=1022.008,110.766,-110.441,167.644,50.089,159.287
C03163=1022.002,110.517,-110.422,167.641,50.095,159.287
C03164=1021.997,110.268,-110.403,167.638,50.101,159.288
C03165=1021.992,110.018,-110.385,167.635,50.106,159.289
C03166=1021.986,109.769,-110.366,167.632,50.112,159.289
C03167=1021.980,109.520,-110.347,167.629,50.118,159.290
C03168=1021.975,109.271,-110.328,167.626,50.124,159.291
C03169=1021.969,109.021,-110.310,167.624,50.129,159.291
C03170=1021.964,108.772,-110.291,167.621,50.135,159.292
C03171=1021.958,108.523,-110.272,167.618,50.141,159.293
C03172=1021.951,108.273,-110.253,167.616,50.146,159.293
C03173=1021.946,107.992,-110.232,167.612,50.153,159.294
C03174=1021.940,107.716,-110.211,167.609,50.159,159.295
C03175=1021.933,107.441,-110.191,167.606,50.165,159.295
C03176=1021.927,107.166,-110.170,167.603,50.172,159.296
C03177=1021.920,106.890,-110.150,167.599,50.178,159.297
C03178=1021.915,106.641,-110.131,167.597,50.184,159.297
C03179=1021.910,106.392,-110.112,167.595,50.189,159.298
C03180=1021.904,106.143,-110.095,167.592,50.195,159.299
C03181=1021.898,105.893,-110.075,167.589,50.201,159.300
C03182=1021.892,105.644,-110.057,167.586,50.206,159.300
C03183=1021.887,105.395,-110.039,167.583,50.212,159.301
C03184=1021.882,105.145,-110.019,167.580,50.218,159.301
C03185=1021.876,104.897,-110.001,167.577,50.224,159.302
C03186=1021.870,104.647,-109.983,167.574,50.229,159.303
C03187=1021.864,104.399,-109.964,167.573,50.235,159.304
C03188=1021.859,104.149,-109.946,167.570,50.240,159.304
C03189=1021.854,103.900,-109.927,167.567,50.246,159.305
C03190=1021.848,103.651,-109.908,167.564,50.252,159.305
C03191=1021.842,103.401,-109.890,167.561,50.258,159.306
C03192=1021.837,103.152,-109.871,167.558,50.264,159.307
C03193=1021.831,102.902,-109.853,167.555,50.269,159.307
C03194=1021.826,102.653,-109.834,167.553,50.274,159.308
C03195=1021.820,102.404,-109.816,167.550,50.280,159.309
C03196=1021.815,102.155,-109.797,167.547,50.286,159.309
C03197=1021.809,101.906,-109.778,167.544,50.291,159.310
C03198=1021.804,101.656,-109.760,167.542,50.297,159.311
C03199=1021.798,101.407,-109.741,167.539,50.303,159.311
C03200=1021.792,101.158,-109.724,167.537,50.308,159.312
C03201=1021.787,100.909,-109.704,167.534,50.314,159.313
C03202=1021.782,100.659,-109.686,167.531,50.320,159.313
C03203=1021.775,100.410,-109.667,167.528,50.325,159.314
C03204=1021.771,100.161,-109.649,167.525,50.331,159.314
C03205=1021.764,99.912,-109.631,167.522,50.336,159.315
C03206=1021.759,99.662,-109.613,167.520,50.342,159.316
C03207=1021.754,99.413,-109.593,167.517,50.348,159.316
C03208=1021.748,99.164,-109.576,167.514,50.353,159.317
C03209=1021.742,98.914,-109.558,167.512,50.359,159.318
C03210=1021.737,98.665,-109.539,167.509,50.365,159.318
C03211=1021.731,98.416,-109.521,167.506,50.371,159.319
C03212=1021.725,98.167,-109.503,167.503,50.376,159.320
C03213=1021.719,97.917,-109.485,167.500,50.382,159.320
C03214=1021.714,97.668,-109.467,167.498,50.388,159.321
C03215=1021.708,97.418,-109.449,167.495,50.393,159.322
C03216=1021.702,97.170,-109.430,167.493,50.399,159.322
C03217=1021.697,96.920,-109.412,167.490,50.405,159.323
C03218=1021.691,96.671,-109.394,167.487,50.411,159.324
C03219=1021.686,96.422,-109.377,167.484,50.417,159.324
C03220=1021.680,96.172,-109.357,167.481,50.422,159.325
C03221=1021.675,95.923,-109.340,167.478,50.428,159.326
C03222=1021.668,95.674,-109.322,167.476,50.434,159.326
C03223=1021.664,95.424,-109.304,167.474,50.439,159.327
C03224=1021.657,95.175,-109.285,167.471,50.445,159.328
C03225=1021.652,94.926,-109.268,167.468,50.451,159.328
C03226=1021.647,94.677,-109.249,167.465,50.457,159.329
C03227=1021.641,94.427,-109.231,167.462,50.462,159.329
C03228=1021.635,94.179,-109.213,167.460,50.468,159.330
C03229=1021.629,93.929,-109.195,167.457,50.474,159.331
C03230=1021.624,93.679,-109.177,167.455,50.479,159.332
C03231=1021.618,93.430,-109.159,167.452,50.485,159.332
C03232=1021.612,93.181,-109.141,167.449,50.491,159.333
C03233=1021.607,92.932,-109.123,167.446,50.497,159.333
C03234=1021.601,92.682,-109.105,167.444,50.502,159.334
C03235=1021.596,92.433,-109.087,167.441,50.507,159.335
C03236=1021.591,92.184,-109.069,167.438,50.513,159.335
C03237=1021.585,91.934,-109.051,167.435,50.519,159.336
C03238=1021.578,91.651,-109.030,167.433,50.525,159.337
C03239=1021.572,91.368,-109.010,167.429,50.532,159.338
C03240=1021.566,91.084,-108.989,167.426,50.538,159.338
C03241=1021.559,90.801,-108.969,167.423,50.545,159.339
C03242=1021.554,90.552,-108.951,167.420,50.551,159.340
C03243=1021.548,90.303,-108.933,167.418,50.556,159.340
C03244=1021.542,90.053,-108.915,167.415,50.562,159.341
C03245=1021.537,89.804,-108.897,167.413,50.568,159.342
C03246=1021.532,89.555,-108.880,167.409,50.573,159.342
C03247=1021.526,89.305,-108.862,167.406,50.579,159.343
C03248=1021.521,89.056,-108.844,167.405,50.584,159.343
C03249=1021.515,88.807,-108.826,167.402,50.590,159.344
C03250=1021.509,88.557,-108.808,167.399,50.596,159.345
C03251=1021.503,88.308,-108.791,167.396,50.601,159.345
C03252=1021.497,88.058,-108.773,167.393,50.607,159.346
C03253=1021.491,87.809,-108.756,167.390,50.613,159.347
C03254=1021.486,87.560,-108.738,167.388,50.619,159.347
C03255=1021.480,87.311,-108.720,167.385,50.625,159.348
C03256=1021.474,87.062,-108.703,167.383,50.631,159.349
C03257=1021.469,86.813,-108.685,167.380,50.637,159.350
C03258=1021.463,86.563,-108.667,167.378,50.642,159.350
C03259=1021.457,86.314,-108.650,167.375,50.648,159.351
C03260=1021.452,86.065,-108.632,167.372,50.654,159.351
C03261=1021.446,85.815,-108.615,167.369,50.660,159.352
C03262=1021.440,85.565,-108.597,167.366,50.666,159.353
C03263=1021.435,85.316,-108.580,167.365,50.671,159.354
C03264=1021.429,85.067,-108.562,167.362,50.677,159.354
C03265=1021.423,84.818,-108.544,167.358,50.682,159.355
C03266=1021.418,84.569,-108.527,167.356,50.688,159.355
C03267=1021.412,84.319,-108.509,167.353,50.694,159.356
C03268=1021.407,84.070,-108.491,167.350,50.700,159.357
C03269=1021.401,83.820,-108.474,167.348,50.705,159.357
C03270=1021.395,83.571,-108.457,167.345,50.711,159.358
C03271=1021.390,83.322,-108.439,167.343,50.717,159.359
C03272=1021.384,83.072,-108.421,167.340,50.723,159.359
C03273=1021.378,82.823,-108.404,167.337,50.728,159.360
C03274=1021.373,82.574,-108.386,167.334,50.734,159.360
C03275=1021.367,82.325,-108.369,167.332,50.740,159.361
C03276=1021.361,82.075,-108.351,167.329,50.745,159.362
C03277=1021.356,81.826,-108.334,167.327,50.751,159.363
C03278=1021.350,81.577,-108.316,167.324,50.757,159.363
C03279=1021.345,81.328,-108.299,167.321,50.763,159.364
C03280=1021.339,81.078,-108.282,167.319,50.768,159.365
C03281=1021.333,80.828,-108.264,167.316,50.774,159.365
C03282=1021.328,80.579,-108.246,167.313,50.779,159.366
C03283=1021.322,80.330,-108.229,167.310,50.785,159.366
C03284=1021.317,80.081,-108.212,167.307,50.791,159.367
C03285=1021.311,79.831,-108.194,167.306,50.797,159.368
C03286=1021.305,79.582,-108.176,167.303,50.802,159.368
C03287=1021.300,79.333,-108.159,167.300,50.808,159.369
C03288=1021.295,79.083,-108.142,167.297,50.814,159.370
C03289=1021.289,78.834,-108.124,167.294,50.819,159.370
C03290=1021.284,78.585,-108.107,167.292,50.825,159.371
C03291=1021.278,78.335,-108.089,167.289,50.830,159.371
C03292=1021.272,78.086,-108.072,167.287,50.836,159.372
C03293=1021.267,77.836,-108.054,167.284,50.842,159.373
C03294=1021.261,77.587,-108.037,167.282,50.848,159.373
C03295=1021.255,77.338,-108.021,167.279,50.853,159.374
C03296=1021.249,77.088,-108.003,167.276,50.859,159.375
C03297=1021.244,76.839,-107.985,167.273,50.864,159.375
C03298=1021.239,76.590,-107.968,167.270,50.870,159.376
C03299=1021.233,76.341,-107.951,167.268,50.876,159.376
C03300=1021.227,76.091,-107.934,167.266,50.882,159.377
C03301=1021.222,75.842,-107.917,167.263,50.887,159.378
C03302=1021.215,75.559,-107.897,167.260,50.894,159.379
C03303=1021.209,75.275,-107.878,167.257,50.901,159.379
C03304=1021.202,74.992,-107.859,167.253,50.907,159.380
C03305=1021.196,74.708,-107.839,167.251,50.914,159.381
C03306=1021.190,74.459,-107.822,167.248,50.919,159.381
C03307=1021.184,74.210,-107.805,167.245,50.925,159.382
C03308=1021.179,73.961,-107.788,167.243,50.931,159.383
C03309=1021.173,73.711,-107.771,167.241,50.937,159.384
C03310=1021.167,73.462,-107.754,167.238,50.943,159.384
C03311=1021.161,73.212,-107.737,167.235,50.948,159.385
C03312=1021.156,72.963,-107.719,167.232,50.954,159.385
C03313=1021.150,72.714,-107.703,167.230,50.960,159.386
C03314=1021.144,72.465,-107.685,167.227,50.966,159.387
C03315=1021.139,72.215,-107.669,167.225,50.971,159.387
C03316=1021.133,71.966,-107.652,167.222,50.977,159.388
C03317=1021.128,71.717,-107.635,167.219,50.982,159.389
C03318=1021.122,71.466,-107.618,167.216,50.988,159.389
C03319=1021.116,71.217,-107.600,167.213,50.994,159.390
C03320=1021.110,70.968,-107.584,167.212,51.000,159.391
C03321=1021.105,70.719,-107.566,167.209,51.006,159.391
C03322=1021.099,70.470,-107.550,167.206,51.011,159.392
C03323=1021.094,70.220,-107.533,167.203,51.017,159.393
C03324=1021.088,69.971,-107.515,167.200,51.023,159.393
C03325=1021.082,69.722,-107.499,167.198,51.028,159.394
C03326=1021.077,69.472,-107.482,167.196,51.034,159.394
C03327=1021.071,69.223,-107.465,167.193,51.040,159.395
C03328=1021.066,68.974,-107.449,167.190,51.045,159.396
C03329=1021.060,68.724,-107.432,167.187,51.051,159.396
C03330=1021.055,68.475,-107.414,167.185,51.057,159.397
C03331=1021.049,68.225,-107.398,167.183,51.063,159.398
C03332=1021.044,67.976,-107.381,167.180,51.069,159.398
C03333=1021.037,67.726,-107.364,167.177,51.074,159.399
C03334=1021.032,67.477,-107.347,167.174,51.080,159.399
C03335=1021.026,67.227,-107.331,167.172,51.085,159.400
C03336=1021.020,66.978,-107.314,167.169,51.091,159.401
C03337=1021.014,66.729,-107.297,167.167,51.097,159.401
C03338=1021.009,66.479,-107.280,167.164,51.103,159.402
C03339=1021.003,66.230,-107.264,167.161,51.109,159.403
C03340=1020.998,65.980,-107.247,167.158,51.115,159.403
C03341=1020.992,65.731,-107.231,167.156,51.120,159.404
C03342=1020.986,65.482,-107.214,167.154,51.126,159.405
C03343=1020.980,65.233,-107.197,167.151,51.132,159.405
C03344=1020.974,64.983,-107.180,167.148,51.137,159.406
C03345=1020.969,64.734,-107.164,167.145,51.143,159.406
C03346=1020.963,64.484,-107.147,167.143,51.148,159.407
C03347=1020.958,64.235,-107.130,167.140,51.154,159.408
C03348=1020.952,63.986,-107.113,167.138,51.160,159.408
C03349=1020.946,63.736,-107.097,167.135,51.166,159.409
C03350=1020.941,63.487,-107.080,167.132,51.172,159.410
C03351=1020.935,63.237,-107.064,167.130,51.177,159.411
C03352=1020.929,62.988,-107.047,167.127,51.183,159.411
C03353=1020.923,62.738,-107.031,167.124,51.188,159.412
C03354=1020.918,62.489,-107.015,167.122,51.195,159.412
C03355=1020.912,62.240,-106.999,167.119,51.201,159.413
C03356=1020.906,61.990,-106.982,167.117,51.207,159.414
C03357=1020.900,61.741,-106.965,167.114,51.213,159.414
C03358=1020.894,61.491,-106.949,167.111,51.219,159.415
C03359=1020.889,61.242,-106.933,167.108,51.224,159.416
C03360=1020.883,60.993,-106.917,167.107,51.230,159.416
C03361=1020.877,60.743,-106.900,167.104,51.236,159.417
C03362=1020.871,60.494,-106.884,167.101,51.242,159.418
C03363=1020.865,60.245,-106.868,167.098,51.248,159.418
C03364=1020.859,59.995,-106.852,167.095,51.254,159.419
C03365=1020.854,59.746,-106.835,167.093,51.259,159.420
C03366=1020.847,59.462,-106.817,167.090,51.266,159.420
C03367=1020.840,59.178,-106.798,167.087,51.272,159.421
C03368=1020.833,58.896,-106.780,167.084,51.279,159.422
C03369=1020.828,58.612,-106.762,167.081,51.286,159.422
C03370=1020.822,58.363,-106.746,167.078,51.292,159.423
C03371=1020.816,58.114,-106.729,167.075,51.298,159.424
C03372=1020.810,57.864,-106.713,167.073,51.303,159.424
C03373=1020.804,57.615,-106.697,167.071,51.309,159.425
C03374=1020.799,57.365,-106.681,167.068,51.315,159.426
C03375=1020.793,57.115,-106.664,167.065,51.321,159.426
C03376=1020.787,56.866,-106.648,167.062,51.326,159.427
C03377=1020.781,56.617,-106.632,167.059,51.332,159.428
C03378=1020.775,56.367,-106.616,167.057,51.338,159.428
C03379=1020.770,56.119,-106.600,167.055,51.343,159.429
C03380=1020.764,55.869,-106.584,167.052,51.349,159.430
C03381=1020.758,55.619,-106.568,167.049,51.355,159.430
C03382=1020.753,55.370,-106.551,167.047,51.361,159.431
C03383=1020.747,55.120,-106.535,167.044,51.367,159.431
C03384=1020.741,54.871,-106.519,167.041,51.373,159.432
C03385=1020.735,54.622,-106.502,167.040,51.378,159.433
C03386=1020.729,54.372,-106.487,167.036,51.384,159.433
C03387=1020.724,54.123,-106.471,167.034,51.390,159.434
C03388=1020.718,53.874,-106.455,167.031,51.395,159.435
C03389=1020.712,53.624,-106.438,167.028,51.401,159.435
C03390=1020.706,53.374,-106.423,167.025,51.407,159.436
C03391=1020.701,53.125,-106.406,167.024,51.413,159.437
C03392=1020.695,52.875,-106.390,167.021,51.418,159.437
C03393=1020.690,52.627,-106.374,167.018,51.424,159.438
C03394=1020.684,52.377,-106.358,167.015,51.430,159.438
C03395=1020.678,52.127,-106.342,167.012,51.436,159.439
C03396=1020.672,51.878,-106.326,167.011,51.441,159.440
C03397=1020.666,51.629,-106.310,167.008,51.447,159.440
C03398=1020.661,51.379,-106.294,167.005,51.452,159.441
C03399=1020.655,51.130,-106.278,167.002,51.458,159.441
C03400=1020.650,50.880,-106.261,166.999,51.464,159.442
C03401=1020.644,50.631,-106.245,166.998,51.470,159.443
C03402=1020.639,50.381,-106.229,166.994,51.475,159.443
C03403=1020.633,50.132,-106.214,166.992,51.481,159.444
C03404=1020.627,49.883,-106.197,166.989,51.487,159.444
C03405=1020.622,49.633,-106.182,166.986,51.493,159.445
C03406=1020.616,49.384,-106.166,166.985,51.498,159.446
C03407=1020.610,49.134,-106.149,166.981,51.504,159.446
C03408=1020.605,48.885,-106.134,166.979,51.510,159.447
C03409=1020.599,48.636,-106.118,166.976,51.516,159.448
C03410=1020.594,48.386,-106.101,166.974,51.520,159.448
C03411=1020.588,48.136,-106.085,166.971,51.526,159.449
C03412=1020.583,47.887,-106.070,166.968,51.532,159.449
C03413=1020.577,47.638,-106.053,166.966,51.538,159.450
C03414=1020.571,47.388,-106.038,166.964,51.543,159.451
C03415=1020.565,47.139,-106.022,166.961,51.549,159.451
C03416=1020.560,46.890,-106.006,166.958,51.555,159.452
C03417=1020.554,46.640,-105.990,166.955,51.560,159.452
C03418=1020.548,46.391,-105.974,166.952,51.566,159.453
C03419=1020.543,46.142,-105.959,166.951,51.572,159.454
C03420=1020.537,45.892,-105.942,166.947,51.577,159.454
C03421=1020.532,45.642,-105.926,166.945,51.583,159.455
C03422=1020.526,45.393,-105.910,166.942,51.589,159.455
C03423=1020.521,45.143,-105.895,166.940,51.594,159.456
C03424=1020.515,44.894,-105.879,166.937,51.600,159.457
C03425=1020.509,44.645,-105.862,166.934,51.605,159.457
C03426=1020.504,44.395,-105.847,166.932,51.610,159.458
C03427=1020.498,44.146,-105.831,166.930,51.616,159.458
C03428=1020.493,43.896,-105.815,166.927,51.622,159.459
C03429=1020.487,43.647,-105.799,166.924,51.627,159.459
C03430=1020.481,43.363,-105.781,166.921,51.634,159.460
C03431=1020.474,43.080,-105.763,166.919,51.640,159.461
C03432=1020.469,42.796,-105.746,166.915,51.646,159.461
C03433=1020.463,42.512,-105.727,166.913,51.653,159.462
C03434=1020.456,42.263,-105.712,166.910,51.658,159.463
C03435=1020.450,42.013,-105.696,166.907,51.664,159.463
C03436=1020.445,41.764,-105.681,166.904,51.670,159.464
C03437=1020.439,41.515,-105.665,166.902,51.676,159.465
C03438=1020.434,41.265,-105.649,166.899,51.681,159.465
C03439=1020.428,41.016,-105.635,166.897,51.687,159.466
C03440=1020.422,40.767,-105.618,166.894,51.693,159.466
C03441=1020.417,40.517,-105.603,166.891,51.699,159.467
C03442=1020.411,40.267,-105.588,166.889,51.704,159.468
C03443=1020.405,40.018,-105.571,166.886,51.710,159.468
C03444=1020.400,39.769,-105.557,166.884,51.716,159.469
C03445=1020.394,39.519,-105.541,166.881,51.721,159.469
C03446=1020.388,39.270,-105.525,166.878,51.727,159.470
C03447=1020.383,39.020,-105.510,166.876,51.732,159.471
C03448=1020.377,38.770,-105.494,166.874,51.738,159.471
C03449=1020.371,38.522,-105.479,166.870,51.744,159.472
C03450=1020.366,38.272,-105.463,166.868,51.749,159.472
C03451=1020.360,38.022,-105.448,166.865,51.755,159.473
C03452=1020.355,37.773,-105.433,166.863,51.760,159.474
C03453=1020.349,37.524,-105.416,166.860,51.766,159.474
C03454=1020.343,37.274,-105.402,166.858,51.772,159.475
C03455=1020.337,37.025,-105.386,166.854,51.778,159.475
C03456=1020.332,36.775,-105.371,166.853,51.783,159.476
C03457=1020.327,36.525,-105.356,166.850,51.789,159.477
C03458=1020.320,36.276,-105.340,166.847,51.794,159.477
C03459=1020.314,36.026,-105.324,166.844,51.800,159.478
C03460=1020.309,35.777,-105.310,166.842,51.806,159.478
C03461=1020.303,35.527,-105.294,166.839,51.812,159.479
C03462=1020.297,35.279,-105.280,166.837,51.817,159.480
C03463=1020.292,35.029,-105.264,166.834,51.823,159.480
C03464=1020.287,34.779,-105.249,166.831,51.829,159.481
C03465=1020.280,34.530,-105.234,166.829,51.835,159.481
C03466=1020.275,34.280,-105.219,166.826,51.840,159.482
C03467=1020.269,34.031,-105.204,166.823,51.846,159.482
C03468=1020.263,33.781,-105.188,166.820,51.852,159.483
C03469=1020.257,33.532,-105.173,166.819,51.858,159.484
C03470=1020.251,33.282,-105.158,166.816,51.863,159.484
C03471=1020.246,33.033,-105.143,166.813,51.869,159.485
C03472=1020.240,32.784,-105.127,166.810,51.875,159.486
C03473=1020.234,32.535,-105.113,166.807,51.881,159.486
C03474=1020.229,32.285,-105.097,166.805,51.886,159.487
C03475=1020.223,32.035,-105.082,166.803,51.892,159.487
C03476=1020.217,31.786,-105.067,166.800,51.898,159.488
C03477=1020.212,31.536,-105.052,166.797,51.903,159.488
C03478=1020.206,31.287,-105.037,166.794,51.909,159.489
C03479=1020.201,31.037,-105.022,166.792,51.915,159.490
C03480=1020.194,30.788,-105.007,166.790,51.920,159.490
C03481=1020.189,30.539,-104.992,166.787,51.926,159.491
C03482=1020.183,30.289,-104.977,166.784,51.932,159.492
C03483=1020.178,30.040,-104.962,166.781,51.937,159.492
C03484=1020.171,29.790,-104.947,166.778,51.943,159.493
C03485=1020.166,29.541,-104.932,166.776,51.948,159.493
C03486=1020.160,29.291,-104.917,166.774,51.954,159.494
C03487=1020.155,29.042,-104.901,166.771,51.960,159.494
C03488=1020.149,28.792,-104.886,166.768,51.965,159.495
C03489=1020.143,28.543,-104.871,166.765,51.971,159.495
C03490=1020.138,28.292,-104.856,166.764,51.977,159.496
C03491=1020.132,28.043,-104.842,166.761,51.982,159.497
C03492=1020.127,27.793,-104.826,166.758,51.988,159.497
C03493=1020.121,27.544,-104.812,166.755,51.993,159.498
C03494=1020.115,27.261,-104.795,166.752,52.000,159.499
C03495=1020.108,26.977,-104.778,166.749,52.007,159.499
C03496=1020.101,26.693,-104.762,166.747,52.013,159.500
C03497=1020.095,26.410,-104.745,166.743,52.020,159.500
C03498=1020.089,26.160,-104.729,166.740,52.026,159.501
C03499=1020.083,25.911,-104.714,166.738,52.030,159.502
C03500=1020.078,25.662,-104.700,166.735,52.036,159.502
C03501=1020.072,25.412,-104.684,166.733,52.042,159.503
C03502=1020.067,25.162,-104.670,166.730,52.048,159.503
C03503=1020.060,24.912,-104.656,166.727,52.054,159.504
C03504=1020.054,24.664,-104.641,166.724,52.060,159.504
C03505=1020.049,24.413,-104.626,166.721,52.065,159.505
C03506=1020.043,24.164,-104.612,166.720,52.071,159.506
C03507=1020.037,23.915,-104.597,166.717,52.077,159.506
C03508=1020.032,23.665,-104.581,166.714,52.082,159.507
C03509=1020.026,23.415,-104.568,166.711,52.088,159.507
C03510=1020.021,23.167,-104.553,166.709,52.094,159.508
C03511=1020.014,22.917,-104.538,166.706,52.099,159.508
C03512=1020.009,22.667,-104.524,166.704,52.105,159.509
C03513=1020.003,22.417,-104.509,166.701,52.111,159.510
C03514=1019.997,22.168,-104.494,166.698,52.116,159.510
C03515=1019.993,21.918,-104.480,166.696,52.122,159.511
C03516=1019.986,21.669,-104.465,166.692,52.127,159.511
C03517=1019.980,21.420,-104.450,166.690,52.133,159.512
C03518=1019.975,21.170,-104.436,166.688,52.139,159.513
C03519=1019.969,20.920,-104.421,166.685,52.144,159.513
C03520=1019.963,20.671,-104.406,166.682,52.150,159.514
C03521=1019.958,20.422,-104.392,166.679,52.156,159.514
C03522=1019.952,20.172,-104.377,166.677,52.162,159.515
C03523=1019.947,19.923,-104.362,166.675,52.167,159.515
C03524=1019.941,19.673,-104.348,166.672,52.173,159.516
C03525=1019.935,19.424,-104.333,166.669,52.178,159.516
C03526=1019.930,19.174,-104.319,166.666,52.184,159.517
C03527=1019.924,18.925,-104.304,166.664,52.190,159.518
C03528=1019.918,18.675,-104.290,166.661,52.195,159.518
C03529=1019.912,18.426,-104.275,166.659,52.201,159.519
C03530=1019.907,18.176,-104.262,166.656,52.206,159.519
C03531=1019.900,17.926,-104.247,166.653,52.212,159.520
C03532=1019.895,17.677,-104.233,166.651,52.218,159.520
C03533=1019.890,17.427,-104.218,166.648,52.224,159.521
C03534=1019.884,17.177,-104.203,166.645,52.230,159.521
C03535=1019.878,16.928,-104.189,166.643,52.234,159.522
C03536=1019.873,16.679,-104.175,166.640,52.241,159.523
C03537=1019.867,16.430,-104.160,166.637,52.246,159.523
C03538=1019.861,16.179,-104.146,166.635,52.252,159.524
C03539=1019.855,15.930,-104.132,166.632,52.258,159.524
C03540=1019.849,15.681,-104.118,166.629,52.263,159.525
C03541=1019.844,15.432,-104.102,166.627,52.269,159.526
C03542=1019.838,15.181,-104.088,166.624,52.274,159.526
C03543=1019.833,14.932,-104.074,166.622,52.280,159.527
C03544=1019.827,14.683,-104.060,166.618,52.285,159.527
C03545=1019.822,14.433,-104.046,166.616,52.291,159.528
C03546=1019.815,14.184,-104.031,166.613,52.297,159.528
C03547=1019.810,13.934,-104.017,166.611,52.302,159.529
C03548=1019.804,13.684,-104.003,166.608,52.308,159.529
C03549=1019.798,13.436,-103.989,166.606,52.314,159.530
C03550=1019.792,13.185,-103.974,166.602,52.319,159.530
C03551=1019.787,12.936,-103.961,166.600,52.325,159.531
C03552=1019.781,12.687,-103.946,166.597,52.331,159.531
C03553=1019.776,12.437,-103.932,166.594,52.336,159.532
C03554=1019.770,12.187,-103.918,166.592,52.343,159.533
C03555=1019.764,11.937,-103.904,166.588,52.348,159.533
C03556=1019.758,11.689,-103.890,166.587,52.354,159.534
C03557=1019.752,11.439,-103.876,166.584,52.360,159.534
C03558=1019.746,11.156,-103.860,166.581,52.366,159.535
C03559=1019.740,10.874,-103.845,166.578,52.372,159.535
C03560=1019.732,10.592,-103.829,166.575,52.379,159.536
C03561=1019.726,10.310,-103.813,166.571,52.385,159.537
C03562=1019.720,10.060,-103.799,166.569,52.391,159.537
C03563=1019.715,9.811,-103.785,166.566,52.396,159.538
C03564=1019.709,9.561,-103.772,166.564,52.402,159.538
C03565=1019.703,9.312,-103.757,166.561,52.408,159.539
C03566=1019.697,9.063,-103.743,166.558,52.414,159.540
C03567=1019.692,8.813,-103.729,166.556,52.420,159.540
C03568=1019.686,8.563,-103.715,166.552,52.425,159.541
C03569=1019.680,8.313,-103.701,166.550,52.431,159.541
C03570=1019.674,8.064,-103.688,166.547,52.437,159.542
C03571=1019.669,7.814,-103.674,166.545,52.442,159.542
C03572=1019.663,7.566,-103.659,166.542,52.448,159.543
C03573=1019.657,7.316,-103.646,166.540,52.454,159.543
C03574=1019.652,7.066,-103.632,166.537,52.459,159.544
C03575=1019.645,6.816,-103.618,166.534,52.465,159.544
C03576=1019.640,6.567,-103.604,166.531,52.470,159.545
